// TIA Portal V20 program export: 1 tag tables, 5 data types, 30 data blocks, 9 code blocks (in call order from the OBs), 26 instance data blocks

VAR_GLOBAL   // PLC tag table "CentralFunctions"
END_VAR

TYPE "typeEmMotorStarterInterface"
// stored: Access Published
   STRUCT
      EMmotorstarter : Array[0.."NO_OF_EM"] of "typeMotorStarterInterface";
   END_STRUCT;
END_TYPE

TYPE "typeEt200SpMotorstarterInterfaceHmi"
// stored: Access Published
   STRUCT
      et200SpMotorstarterReadValue : Bool;   // read Value of MotorStarter
      et200SpNumberOfMotorstarters { ExternalWritable := 'False'} : USInt;   // Number of Motor Starters
      et200SpUnitMotorstarter : USInt := 1;   // Unit selected
      et200SpEMMotorstarter : USInt := 0;   // Equipment Module selected
      et200SpMotorstarterCurrent : Array[0.."NO_OF_ET200SPMOTORSTARTER"] of Real;   // Aktuelle Werte / Current values
      et200SpMotorstarterInputs : Array[0.."NO_OF_ET200SPMOTORSTARTER"] of "LSicar_typeMotorstarterIn";   // Motorstarter Data Inputs HMI
      et200SpMotorstarterOutputs : Array[0.."NO_OF_ET200SPMOTORSTARTER"] of "LSicar_typeMotorstarterOut";   // Motorstarter Data Outputs HMI
   END_STRUCT;
END_TYPE

TYPE "typeMotorStarterInterface"
// stored: Access Published
   STRUCT
      et200SpMotorstarterCurrent : Array[0.."NO_OF_ET200SPMOTORSTARTER"] of Real;   // Aktuelle Werte / Current values
      et200SpMotorstarterInputs : Array[0.."NO_OF_ET200SPMOTORSTARTER"] of "LSicar_typeMotorstarterIn";   // Motorstarter Data Inputs HMI
      et200SpMotorstarterOutputs : Array[0.."NO_OF_ET200SPMOTORSTARTER"] of "LSicar_typeMotorstarterOut";   // Motorstarter Data Outputs HMI
   END_STRUCT;
END_TYPE

TYPE "typeIdentMvHmi"
// stored: Access Published
   STRUCT
      selectedUnit : USInt;
      selectedEM : USInt;
      mvReaderId : USInt;   // MV Reader ID
      numberOfMv : USInt;   // Anzahl der MV Antriebe / Number of used MV readers
      mvReader : Array[0.."NO_OF_MV_IDENT_DEVICES"] of "LSicar_typeIdentInterfaceHmi";   // MV Reader
   END_STRUCT;
END_TYPE

TYPE "typeEMIdentRf"
// stored: Access Published
   STRUCT
      identRfEM : Array[0.."NO_OF_EM"] of "typeIdentRfHmi";
   END_STRUCT;
END_TYPE

DATA_BLOCK "TestTempDB"   // DB502
// stored: MemoryReserve 100
   VAR
      TempBool : Array[0..100] of Bool;
   END_VAR
BEGIN
END_DATA_BLOCK

DATA_BLOCK "Simulation"   // DB203
TITLE = Simulation
// Simulation data
// stored: MemoryReserve 100
   VAR
      simHmiRotaryAxis : Array[0..49] of "LER_typeSimRotaryAxis";
      simHmiLinearAxis : Array[0..49] of "LER_typeSimLinearAxis";
      data : "LAF_typeSimulation";
   END_VAR
BEGIN
   data.simitActive := FALSE;
   data.simulationActiveHmi := TRUE;
   data.showSimulationButtonHmi := TRUE;
END_DATA_BLOCK

DATA_BLOCK "ProdDataInterfaceHmi"   // DB53
TITLE = HMI und Anwender Schnittstelle für Produktionsdaten / HMI and user interface for production data
AUTHOR : SICAR
FAMILY : ProdData
// FUNKTIONSBESCHREIBUNG: 
// Der Baustein beinhaltet alle Informationen zum und vom HMI, sowie die Anwenderschnittstellen für die Produktionsdaten
// Weitere Hinweise: siehe SICAR anwenderdefinierte Dokumentation / SICAR Online-Hilfe.
// DESCRIPTION OF FUNCTIONS:
// stored: MemoryReserve 100
   VAR RETAIN
      numberOfDataSets : "LSicar_typeNumberOfDataSets";   // Anzahl konfigurierter Datensätze / Number of configured data sets
   END_VAR
   VAR
      colorCodeLimitSummary : UInt := 0;   // Gesamt Status Grenzwerte / Overall status Limit values
      colorCodeLimitSelButton : Array[0..8] of UInt;   // Farbcode für Datensatz Anwahl Button (Grenzwerte) / Color code for data set select button (Limit values)
   END_VAR
   VAR RETAIN
      limitValueDataSetSel : Int := 1;   // Angwaehlter Datensatz Grenzwerte / selected data set limit values
      limitDataSet : Array[0.."NO_DATASETS_LIMITVALUES"] of "LSicar_typeLimitValue";   // Datensätze Grenzwerte / Data sets limit .values
      cycleTimerDataSetSel : Int := 1;   // Angewaehlter Datensatz Taktzeiten / selected data set cycle timer
      cycleTimerDataSet : Array[0.."NO_DATASETS_CYCLETIMER"] of "LSicar_typeCycleTimer";   // Datensätze Taktzeiten / Data sets cycle timer
      counterDataSetSel : Int := 1;   // Angewählter Datensatz Zaehler / selected data set counter
      counterDataSet : Array[0.."NO_DATASETS_COUNTER"] of "LSicar_typeCounter";   // Datensätze Zähler / Data sets counter
      shiftCounterDataSetSel : Int := 1;   // Angewaehlter Datensatz Schichtzaehler / selected data set shift counter
      shiftCounterDataSet : Array[0.."NO_DATASETS_SHIFTCOUNTER"] of "LSicar_typeShiftCounter";   // Datensätze Schichtzähler / Data sets shift counter
      shiftCountOeeDataSetSel : Int := 1;   // Angewaehlter Datensatz OEE / selected data set OEE
      shiftCounterOeeDataSet : Array[0.."NO_DATASETS_SHIFTCOUNTER"] of "LSicar_typeShiftCounterOee";   // Datensätze Schichtzähler OEE / Data sets shift counter OEE
   END_VAR
BEGIN
   numberOfDataSets.limitValues := 2;
   numberOfDataSets.cycleTimer := 2;
   numberOfDataSets."counter" := 2;
   numberOfDataSets.shiftCounter := 2;
   colorCodeLimitSelButton[0..8] := 0;
   limitDataSet[0].targetValue[0..10] := 0;
   limitDataSet[1].targetValue[0..10] := 0;
   limitDataSet[2].targetValue[0..10] := 0;
   limitDataSet[0].prewarnValue[0..10] := 0;
   limitDataSet[1].prewarnValue[0..10] := 0;
   limitDataSet[2].prewarnValue[0..10] := 0;
   limitDataSet[0].remainValue[0..10] := 0;
   limitDataSet[1].remainValue[0..10] := 0;
   limitDataSet[2].remainValue[0..10] := 0;
   limitDataSet[0].control[0..10].count := FALSE;
   limitDataSet[1].control[0..10].count := FALSE;
   limitDataSet[2].control[0..10].count := FALSE;
   limitDataSet[0].control[0..10].set := FALSE;
   limitDataSet[1].control[0..10].set := FALSE;
   limitDataSet[2].control[0..10].set := FALSE;
   limitDataSet[0].control[0..10].prewarn := FALSE;
   limitDataSet[1].control[0..10].prewarn := FALSE;
   limitDataSet[2].control[0..10].prewarn := FALSE;
   limitDataSet[0].control[0..10].alarm := FALSE;
   limitDataSet[1].control[0..10].alarm := FALSE;
   limitDataSet[2].control[0..10].alarm := FALSE;
   limitDataSet[0].textListValue[0..10] := 0;
   limitDataSet[1].textListValue[0..10] := 0;
   limitDataSet[2].textListValue[0..10] := 0;
   limitDataSet[0..2].userInterfaceVisibility := 16#0000_0000;
   limitDataSet[0].colorCodeAlarmPrewarn[0..10] := 0;
   limitDataSet[1].colorCodeAlarmPrewarn[0..10] := 0;
   limitDataSet[2].colorCodeAlarmPrewarn[0..10] := 0;
   limitDataSet[0..2].indexSelectedLimitValue := 0;
   limitDataSet[0..2].divButton := 16#00;
   limitDataSet[0..2].visibility := 16#0000_0000;
   cycleTimerDataSet[0].targetValue[0..20] := 0;
   cycleTimerDataSet[1].targetValue[0..20] := 0;
   cycleTimerDataSet[2].targetValue[0..20] := 0;
   cycleTimerDataSet[0].currentValue[0..20] := 0;
   cycleTimerDataSet[1].currentValue[0..20] := 0;
   cycleTimerDataSet[2].currentValue[0..20] := 0;
   cycleTimerDataSet[0].averageValue[0..20] := 0;
   cycleTimerDataSet[1].averageValue[0..20] := 0;
   cycleTimerDataSet[2].averageValue[0..20] := 0;
   cycleTimerDataSet[0].counts[0..20] := 0;
   cycleTimerDataSet[1].counts[0..20] := 0;
   cycleTimerDataSet[2].counts[0..20] := 0;
   cycleTimerDataSet[0].measureActive[0..20] := 0;
   cycleTimerDataSet[1].measureActive[0..20] := 0;
   cycleTimerDataSet[2].measureActive[0..20] := 0;
   cycleTimerDataSet[0].control[0..20].run := FALSE;
   cycleTimerDataSet[1].control[0..20].run := FALSE;
   cycleTimerDataSet[2].control[0..20].run := FALSE;
   cycleTimerDataSet[0].control[0..20].hold := FALSE;
   cycleTimerDataSet[1].control[0..20].hold := FALSE;
   cycleTimerDataSet[2].control[0..20].hold := FALSE;
   cycleTimerDataSet[0].control[0..20].reset := FALSE;
   cycleTimerDataSet[1].control[0..20].reset := FALSE;
   cycleTimerDataSet[2].control[0..20].reset := FALSE;
   cycleTimerDataSet[0].textListValue[0..20] := 0;
   cycleTimerDataSet[1].textListValue[0..20] := 0;
   cycleTimerDataSet[2].textListValue[0..20] := 0;
   cycleTimerDataSet[0..2].userInterfaceVisibility := 16#0000_0000;
   cycleTimerDataSet[0..2].resetAverageAllExt := FALSE;
   cycleTimerDataSet[0..2].indexSelectedTimer := 0;
   cycleTimerDataSet[0..2].divButton := 16#00;
   cycleTimerDataSet[0..2].visibility := 16#0000_0000;
   counterDataSet[0].currentValue[0..20] := 0;
   counterDataSet[1].currentValue[0..20] := 0;
   counterDataSet[2].currentValue[0..20] := 0;
   counterDataSet[0].control[0..20].countUp := FALSE;
   counterDataSet[1].control[0..20].countUp := FALSE;
   counterDataSet[2].control[0..20].countUp := FALSE;
   counterDataSet[0].control[0..20].countDown := FALSE;
   counterDataSet[1].control[0..20].countDown := FALSE;
   counterDataSet[2].control[0..20].countDown := FALSE;
   counterDataSet[0].control[0..20].reset := FALSE;
   counterDataSet[1].control[0..20].reset := FALSE;
   counterDataSet[2].control[0..20].reset := FALSE;
   counterDataSet[0].textListValue[0..20] := 0;
   counterDataSet[1].textListValue[0..20] := 0;
   counterDataSet[2].textListValue[0..20] := 0;
   counterDataSet[0].userInterfaceVisibility := 16#0000_0000;
   counterDataSet[1].userInterfaceVisibility := 16#0000_0007;
   counterDataSet[2].userInterfaceVisibility := 16#0000_0003;
   counterDataSet[0..2].resetAllExt := FALSE;
   counterDataSet[0..2].indexSelectedCounter := 0;
   counterDataSet[0..2].divButton := 16#00;
   counterDataSet[0..2].visibility := 16#0000_0000;
   shiftCounterDataSet[0].currentShiftValue.partsTarget[0..10] := 0;
   shiftCounterDataSet[1].currentShiftValue.partsTarget[0..10] := 0;
   shiftCounterDataSet[2].currentShiftValue.partsTarget[0..10] := 0;
   shiftCounterDataSet[0].currentShiftValue.partsCurrent[0..10] := 0;
   shiftCounterDataSet[1].currentShiftValue.partsCurrent[0..10] := 0;
   shiftCounterDataSet[2].currentShiftValue.partsCurrent[0..10] := 0;
   shiftCounterDataSet[0].previousShiftValue.partsTarget[0..10] := 0;
   shiftCounterDataSet[1].previousShiftValue.partsTarget[0..10] := 0;
   shiftCounterDataSet[2].previousShiftValue.partsTarget[0..10] := 0;
   shiftCounterDataSet[0].previousShiftValue.partsCurrent[0..10] := 0;
   shiftCounterDataSet[1].previousShiftValue.partsCurrent[0..10] := 0;
   shiftCounterDataSet[2].previousShiftValue.partsCurrent[0..10] := 0;
   shiftCounterDataSet[0].penultimateShiftValue.partsTarget[0..10] := 0;
   shiftCounterDataSet[1].penultimateShiftValue.partsTarget[0..10] := 0;
   shiftCounterDataSet[2].penultimateShiftValue.partsTarget[0..10] := 0;
   shiftCounterDataSet[0].penultimateShiftValue.partsCurrent[0..10] := 0;
   shiftCounterDataSet[1].penultimateShiftValue.partsCurrent[0..10] := 0;
   shiftCounterDataSet[2].penultimateShiftValue.partsCurrent[0..10] := 0;
   shiftCounterDataSet[0].countPartsCurrent[0..10] := FALSE;
   shiftCounterDataSet[1].countPartsCurrent[0..10] := FALSE;
   shiftCounterDataSet[2].countPartsCurrent[0..10] := FALSE;
   shiftCounterDataSet[0].textListValue[0..10] := 0;
   shiftCounterDataSet[1].textListValue[0..10] := 0;
   shiftCounterDataSet[2].textListValue[0..10] := 0;
   shiftCounterDataSet[0..2].userInterfaceVisibility := 16#0000_0000;
   shiftCounterDataSet[0..2].resetAllExt := FALSE;
   shiftCounterDataSet[0..2].divButton := 16#00;
   shiftCounterDataSet[0..2].visibility := 16#0000_0000;
   shiftCounterOeeDataSet[0].currentShiftValue.oee[0..10] := 0.0;
   shiftCounterOeeDataSet[1].currentShiftValue.oee[0..10] := 0.0;
   shiftCounterOeeDataSet[2].currentShiftValue.oee[0..10] := 0.0;
   shiftCounterOeeDataSet[0].currentShiftValue.trend[0..10] := 0;
   shiftCounterOeeDataSet[1].currentShiftValue.trend[0..10] := 0;
   shiftCounterOeeDataSet[2].currentShiftValue.trend[0..10] := 0;
   shiftCounterOeeDataSet[0].currentShiftValue.partsTarget[0..10] := 0;
   shiftCounterOeeDataSet[1].currentShiftValue.partsTarget[0..10] := 0;
   shiftCounterOeeDataSet[2].currentShiftValue.partsTarget[0..10] := 0;
   shiftCounterOeeDataSet[0].currentShiftValue.partsCurrent[0..10] := 0;
   shiftCounterOeeDataSet[1].currentShiftValue.partsCurrent[0..10] := 0;
   shiftCounterOeeDataSet[2].currentShiftValue.partsCurrent[0..10] := 0;
   shiftCounterOeeDataSet[0].currentShiftValue.partsCurrentOk[0..10] := 0;
   shiftCounterOeeDataSet[1].currentShiftValue.partsCurrentOk[0..10] := 0;
   shiftCounterOeeDataSet[2].currentShiftValue.partsCurrentOk[0..10] := 0;
   shiftCounterOeeDataSet[0].previousShiftValue.oee[0..10] := 0.0;
   shiftCounterOeeDataSet[1].previousShiftValue.oee[0..10] := 0.0;
   shiftCounterOeeDataSet[2].previousShiftValue.oee[0..10] := 0.0;
   shiftCounterOeeDataSet[0].previousShiftValue.trend[0..10] := 0;
   shiftCounterOeeDataSet[1].previousShiftValue.trend[0..10] := 0;
   shiftCounterOeeDataSet[2].previousShiftValue.trend[0..10] := 0;
   shiftCounterOeeDataSet[0].previousShiftValue.partsTarget[0..10] := 0;
   shiftCounterOeeDataSet[1].previousShiftValue.partsTarget[0..10] := 0;
   shiftCounterOeeDataSet[2].previousShiftValue.partsTarget[0..10] := 0;
   shiftCounterOeeDataSet[0].previousShiftValue.partsCurrent[0..10] := 0;
   shiftCounterOeeDataSet[1].previousShiftValue.partsCurrent[0..10] := 0;
   shiftCounterOeeDataSet[2].previousShiftValue.partsCurrent[0..10] := 0;
   shiftCounterOeeDataSet[0].previousShiftValue.partsCurrentOk[0..10] := 0;
   shiftCounterOeeDataSet[1].previousShiftValue.partsCurrentOk[0..10] := 0;
   shiftCounterOeeDataSet[2].previousShiftValue.partsCurrentOk[0..10] := 0;
   shiftCounterOeeDataSet[0].penultimateShiftValue.oee[0..10] := 0.0;
   shiftCounterOeeDataSet[1].penultimateShiftValue.oee[0..10] := 0.0;
   shiftCounterOeeDataSet[2].penultimateShiftValue.oee[0..10] := 0.0;
   shiftCounterOeeDataSet[0].penultimateShiftValue.trend[0..10] := 0;
   shiftCounterOeeDataSet[1].penultimateShiftValue.trend[0..10] := 0;
   shiftCounterOeeDataSet[2].penultimateShiftValue.trend[0..10] := 0;
   shiftCounterOeeDataSet[0].penultimateShiftValue.partsTarget[0..10] := 0;
   shiftCounterOeeDataSet[1].penultimateShiftValue.partsTarget[0..10] := 0;
   shiftCounterOeeDataSet[2].penultimateShiftValue.partsTarget[0..10] := 0;
   shiftCounterOeeDataSet[0].penultimateShiftValue.partsCurrent[0..10] := 0;
   shiftCounterOeeDataSet[1].penultimateShiftValue.partsCurrent[0..10] := 0;
   shiftCounterOeeDataSet[2].penultimateShiftValue.partsCurrent[0..10] := 0;
   shiftCounterOeeDataSet[0].penultimateShiftValue.partsCurrentOk[0..10] := 0;
   shiftCounterOeeDataSet[1].penultimateShiftValue.partsCurrentOk[0..10] := 0;
   shiftCounterOeeDataSet[2].penultimateShiftValue.partsCurrentOk[0..10] := 0;
   shiftCounterOeeDataSet[0].countPartsCurrent[0..10] := FALSE;
   shiftCounterOeeDataSet[1].countPartsCurrent[0..10] := FALSE;
   shiftCounterOeeDataSet[2].countPartsCurrent[0..10] := FALSE;
   shiftCounterOeeDataSet[0].countPartsCurrentOk[0..10] := FALSE;
   shiftCounterOeeDataSet[1].countPartsCurrentOk[0..10] := FALSE;
   shiftCounterOeeDataSet[2].countPartsCurrentOk[0..10] := FALSE;
   shiftCounterOeeDataSet[0].textListValue[0..10] := 0;
   shiftCounterOeeDataSet[1].textListValue[0..10] := 0;
   shiftCounterOeeDataSet[2].textListValue[0..10] := 0;
   shiftCounterOeeDataSet[0..2].userInterfaceVisibility := 16#0000_0000;
   shiftCounterOeeDataSet[0..2].resetAllExt := FALSE;
   shiftCounterOeeDataSet[0..2].divButton := 16#00;
   shiftCounterOeeDataSet[0..2].visibility := 16#0000_0000;
END_DATA_BLOCK

DATA_BLOCK "ShiftTimesList"   // DB52
TITLE = Shifttimes / Shift times
{ DB_Accessible_From_OPC_UA := 'FALSE' }
AUTHOR : SICAR
FAMILY : Shiftmodel
// Schichtzeiten Liste / Shift times List
// stored: DBAccessibleFromOPCUA false, MemoryReserve 100
   VAR
      list { ExternalAccessible := 'False'; ExternalVisible := 'False'; ExternalWritable := 'False'} : Array[0..10] of "LSicar_typeShiftmodTime1DaySel";   // Schichtmodel Liste / Shiftmodel list
   END_VAR
BEGIN
   list[0..2].listValidFor.sunday := FALSE;
   list[3].listValidFor.sunday := TRUE;
   list[4..10].listValidFor.sunday := FALSE;
   list[0].listValidFor.monday := FALSE;
   list[1..3].listValidFor.monday := TRUE;
   list[4..10].listValidFor.monday := FALSE;
   list[0].listValidFor.tuesday := FALSE;
   list[1..3].listValidFor.tuesday := TRUE;
   list[4..10].listValidFor.tuesday := FALSE;
   list[0].listValidFor.wednesday := FALSE;
   list[1..3].listValidFor.wednesday := TRUE;
   list[4..10].listValidFor.wednesday := FALSE;
   list[0].listValidFor.thursday := FALSE;
   list[1..3].listValidFor.thursday := TRUE;
   list[4..10].listValidFor.thursday := FALSE;
   list[0].listValidFor.friday := FALSE;
   list[1].listValidFor.friday := TRUE;
   list[2].listValidFor.friday := FALSE;
   list[3].listValidFor.friday := TRUE;
   list[4..10].listValidFor.friday := FALSE;
   list[0..2].listValidFor.saturday := FALSE;
   list[3].listValidFor.saturday := TRUE;
   list[4..10].listValidFor.saturday := FALSE;
   list[0].shift[0..3].endCircuitTime := TOD#00:00:00;
   list[1].shift[0].endCircuitTime := TOD#00:00:00;
   list[1].shift[1].endCircuitTime := TOD#05:57:00;
   list[1].shift[2].endCircuitTime := TOD#13:57:00;
   list[1].shift[3].endCircuitTime := TOD#21:57:00;
   list[2].shift[0].endCircuitTime := TOD#00:00:00;
   list[2].shift[1].endCircuitTime := TOD#04:57:00;
   list[2].shift[2].endCircuitTime := TOD#14:27:00;
   list[2].shift[3].endCircuitTime := TOD#00:00:00;
   list[3].shift[0].endCircuitTime := TOD#00:00:00;
   list[3].shift[1].endCircuitTime := TOD#05:57:00;
   list[3].shift[2].endCircuitTime := TOD#14:27:00;
   list[3].shift[3].endCircuitTime := TOD#22:57:00;
   list[4].shift[0..3].endCircuitTime := TOD#00:00:00;
   list[5].shift[0..3].endCircuitTime := TOD#00:00:00;
   list[6].shift[0..3].endCircuitTime := TOD#00:00:00;
   list[7].shift[0..3].endCircuitTime := TOD#00:00:00;
   list[8].shift[0..3].endCircuitTime := TOD#00:00:00;
   list[9].shift[0..3].endCircuitTime := TOD#00:00:00;
   list[10].shift[0..3].endCircuitTime := TOD#00:00:00;
   list[0].shift[0..3].start := TOD#00:00:00;
   list[1].shift[0].start := TOD#00:00:00;
   list[1].shift[1].start := TOD#06:00:00;
   list[1].shift[2].start := TOD#14:00:00;
   list[1].shift[3].start := TOD#22:00:00;
   list[2].shift[0].start := TOD#00:00:00;
   list[2].shift[1].start := TOD#05:00:00;
   list[2].shift[2].start := TOD#14:30:00;
   list[2].shift[3].start := TOD#00:00:00;
   list[3].shift[0].start := TOD#00:00:00;
   list[3].shift[1].start := TOD#06:00:00;
   list[3].shift[2].start := TOD#14:30:00;
   list[3].shift[3].start := TOD#23:00:00;
   list[4].shift[0..3].start := TOD#00:00:00;
   list[5].shift[0..3].start := TOD#00:00:00;
   list[6].shift[0..3].start := TOD#00:00:00;
   list[7].shift[0..3].start := TOD#00:00:00;
   list[8].shift[0..3].start := TOD#00:00:00;
   list[9].shift[0..3].start := TOD#00:00:00;
   list[10].shift[0..3].start := TOD#00:00:00;
   list[0].shift[0].break[0..4].start := TOD#00:00:00;
   list[0].shift[1].break[0..4].start := TOD#00:00:00;
   list[0].shift[2].break[0..4].start := TOD#00:00:00;
   list[0].shift[3].break[0..4].start := TOD#00:00:00;
   list[1].shift[0].break[0..4].start := TOD#00:00:00;
   list[1].shift[1].break[0].start := TOD#00:00:00;
   list[1].shift[1].break[1].start := TOD#08:00:00;
   list[1].shift[1].break[2].start := TOD#10:00:00;
   list[1].shift[1].break[3].start := TOD#12:00:00;
   list[1].shift[1].break[4].start := TOD#00:00:00;
   list[1].shift[2].break[0].start := TOD#00:00:00;
   list[1].shift[2].break[1].start := TOD#16:00:00;
   list[1].shift[2].break[2].start := TOD#18:00:00;
   list[1].shift[2].break[3].start := TOD#20:00:00;
   list[1].shift[2].break[4].start := TOD#00:00:00;
   list[1].shift[3].break[0..1].start := TOD#00:00:00;
   list[1].shift[3].break[2].start := TOD#02:00:00;
   list[1].shift[3].break[3].start := TOD#04:00:00;
   list[1].shift[3].break[4].start := TOD#00:00:00;
   list[2].shift[0].break[0..4].start := TOD#00:00:00;
   list[2].shift[1].break[0].start := TOD#00:00:00;
   list[2].shift[1].break[1].start := TOD#07:00:00;
   list[2].shift[1].break[2].start := TOD#09:00:00;
   list[2].shift[1].break[3].start := TOD#11:00:00;
   list[2].shift[1].break[4].start := TOD#13:00:00;
   list[2].shift[2].break[0].start := TOD#00:00:00;
   list[2].shift[2].break[1].start := TOD#16:30:00;
   list[2].shift[2].break[2].start := TOD#18:30:00;
   list[2].shift[2].break[3].start := TOD#20:30:00;
   list[2].shift[2].break[4].start := TOD#22:00:00;
   list[2].shift[3].break[0..4].start := TOD#00:00:00;
   list[3].shift[0].break[0..4].start := TOD#00:00:00;
   list[3].shift[1].break[0].start := TOD#00:00:00;
   list[3].shift[1].break[1].start := TOD#08:00:00;
   list[3].shift[1].break[2].start := TOD#10:00:00;
   list[3].shift[1].break[3].start := TOD#11:30:00;
   list[3].shift[1].break[4].start := TOD#12:30:00;
   list[3].shift[2].break[0].start := TOD#00:00:00;
   list[3].shift[2].break[1].start := TOD#16:00:00;
   list[3].shift[2].break[2].start := TOD#18:00:00;
   list[3].shift[2].break[3].start := TOD#19:30:00;
   list[3].shift[2].break[4].start := TOD#20:30:00;
   list[3].shift[3].break[0..1].start := TOD#00:00:00;
   list[3].shift[3].break[2].start := TOD#02:00:00;
   list[3].shift[3].break[3].start := TOD#03:30:00;
   list[3].shift[3].break[4].start := TOD#04:30:00;
   list[4].shift[0].break[0..4].start := TOD#00:00:00;
   list[4].shift[1].break[0..4].start := TOD#00:00:00;
   list[4].shift[2].break[0..4].start := TOD#00:00:00;
   list[4].shift[3].break[0..4].start := TOD#00:00:00;
   list[5].shift[0].break[0..4].start := TOD#00:00:00;
   list[5].shift[1].break[0..4].start := TOD#00:00:00;
   list[5].shift[2].break[0..4].start := TOD#00:00:00;
   list[5].shift[3].break[0..4].start := TOD#00:00:00;
   list[6].shift[0].break[0..4].start := TOD#00:00:00;
   list[6].shift[1].break[0..4].start := TOD#00:00:00;
   list[6].shift[2].break[0..4].start := TOD#00:00:00;
   list[6].shift[3].break[0..4].start := TOD#00:00:00;
   list[7].shift[0].break[0..4].start := TOD#00:00:00;
   list[7].shift[1].break[0..4].start := TOD#00:00:00;
   list[7].shift[2].break[0..4].start := TOD#00:00:00;
   list[7].shift[3].break[0..4].start := TOD#00:00:00;
   list[8].shift[0].break[0..4].start := TOD#00:00:00;
   list[8].shift[1].break[0..4].start := TOD#00:00:00;
   list[8].shift[2].break[0..4].start := TOD#00:00:00;
   list[8].shift[3].break[0..4].start := TOD#00:00:00;
   list[9].shift[0].break[0..4].start := TOD#00:00:00;
   list[9].shift[1].break[0..4].start := TOD#00:00:00;
   list[9].shift[2].break[0..4].start := TOD#00:00:00;
   list[9].shift[3].break[0..4].start := TOD#00:00:00;
   list[10].shift[0].break[0..4].start := TOD#00:00:00;
   list[10].shift[1].break[0..4].start := TOD#00:00:00;
   list[10].shift[2].break[0..4].start := TOD#00:00:00;
   list[10].shift[3].break[0..4].start := TOD#00:00:00;
   list[0].shift[0].break[0..4].startCircuitTime := TOD#00:00:00;
   list[0].shift[1].break[0..4].startCircuitTime := TOD#00:00:00;
   list[0].shift[2].break[0..4].startCircuitTime := TOD#00:00:00;
   list[0].shift[3].break[0..4].startCircuitTime := TOD#00:00:00;
   list[1].shift[0].break[0..4].startCircuitTime := TOD#00:00:00;
   list[1].shift[1].break[0].startCircuitTime := TOD#00:00:00;
   list[1].shift[1].break[1].startCircuitTime := TOD#08:02:00;
   list[1].shift[1].break[2].startCircuitTime := TOD#00:00:00;
   list[1].shift[1].break[3].startCircuitTime := TOD#12:02:00;
   list[1].shift[1].break[4].startCircuitTime := TOD#00:00:00;
   list[1].shift[2].break[0].startCircuitTime := TOD#00:00:00;
   list[1].shift[2].break[1].startCircuitTime := TOD#16:02:00;
   list[1].shift[2].break[2].startCircuitTime := TOD#00:00:00;
   list[1].shift[2].break[3].startCircuitTime := TOD#20:02:00;
   list[1].shift[2].break[4].startCircuitTime := TOD#00:00:00;
   list[1].shift[3].break[0].startCircuitTime := TOD#00:00:00;
   list[1].shift[3].break[1].startCircuitTime := TOD#00:02:00;
   list[1].shift[3].break[2].startCircuitTime := TOD#00:00:00;
   list[1].shift[3].break[3].startCircuitTime := TOD#04:02:00;
   list[1].shift[3].break[4].startCircuitTime := TOD#00:00:00;
   list[2].shift[0].break[0..4].startCircuitTime := TOD#00:00:00;
   list[2].shift[1].break[0].startCircuitTime := TOD#00:00:00;
   list[2].shift[1].break[1].startCircuitTime := TOD#07:02:00;
   list[2].shift[1].break[2].startCircuitTime := TOD#00:00:00;
   list[2].shift[1].break[3].startCircuitTime := TOD#11:02:00;
   list[2].shift[1].break[4].startCircuitTime := TOD#13:02:00;
   list[2].shift[2].break[0].startCircuitTime := TOD#00:00:00;
   list[2].shift[2].break[1].startCircuitTime := TOD#16:32:00;
   list[2].shift[2].break[2].startCircuitTime := TOD#00:00:00;
   list[2].shift[2].break[3].startCircuitTime := TOD#20:32:00;
   list[2].shift[2].break[4].startCircuitTime := TOD#22:02:00;
   list[2].shift[3].break[0..4].startCircuitTime := TOD#00:00:00;
   list[3].shift[0].break[0..4].startCircuitTime := TOD#00:00:00;
   list[3].shift[1].break[0..1].startCircuitTime := TOD#00:00:00;
   list[3].shift[1].break[2].startCircuitTime := TOD#10:02:00;
   list[3].shift[1].break[3].startCircuitTime := TOD#00:00:00;
   list[3].shift[1].break[4].startCircuitTime := TOD#12:32:00;
   list[3].shift[2].break[0..1].startCircuitTime := TOD#00:00:00;
   list[3].shift[2].break[2].startCircuitTime := TOD#18:02:00;
   list[3].shift[2].break[3].startCircuitTime := TOD#00:00:00;
   list[3].shift[2].break[4].startCircuitTime := TOD#20:32:00;
   list[3].shift[3].break[0..1].startCircuitTime := TOD#00:00:00;
   list[3].shift[3].break[2].startCircuitTime := TOD#02:02:00;
   list[3].shift[3].break[3..4].startCircuitTime := TOD#00:00:00;
   list[4].shift[0].break[0..4].startCircuitTime := TOD#00:00:00;
   list[4].shift[1].break[0..4].startCircuitTime := TOD#00:00:00;
   list[4].shift[2].break[0..4].startCircuitTime := TOD#00:00:00;
   list[4].shift[3].break[0..4].startCircuitTime := TOD#00:00:00;
   list[5].shift[0].break[0..4].startCircuitTime := TOD#00:00:00;
   list[5].shift[1].break[0..4].startCircuitTime := TOD#00:00:00;
   list[5].shift[2].break[0..4].startCircuitTime := TOD#00:00:00;
   list[5].shift[3].break[0..4].startCircuitTime := TOD#00:00:00;
   list[6].shift[0].break[0..4].startCircuitTime := TOD#00:00:00;
   list[6].shift[1].break[0..4].startCircuitTime := TOD#00:00:00;
   list[6].shift[2].break[0..4].startCircuitTime := TOD#00:00:00;
   list[6].shift[3].break[0..4].startCircuitTime := TOD#00:00:00;
   list[7].shift[0].break[0..4].startCircuitTime := TOD#00:00:00;
   list[7].shift[1].break[0..4].startCircuitTime := TOD#00:00:00;
   list[7].shift[2].break[0..4].startCircuitTime := TOD#00:00:00;
   list[7].shift[3].break[0..4].startCircuitTime := TOD#00:00:00;
   list[8].shift[0].break[0..4].startCircuitTime := TOD#00:00:00;
   list[8].shift[1].break[0..4].startCircuitTime := TOD#00:00:00;
   list[8].shift[2].break[0..4].startCircuitTime := TOD#00:00:00;
   list[8].shift[3].break[0..4].startCircuitTime := TOD#00:00:00;
   list[9].shift[0].break[0..4].startCircuitTime := TOD#00:00:00;
   list[9].shift[1].break[0..4].startCircuitTime := TOD#00:00:00;
   list[9].shift[2].break[0..4].startCircuitTime := TOD#00:00:00;
   list[9].shift[3].break[0..4].startCircuitTime := TOD#00:00:00;
   list[10].shift[0].break[0..4].startCircuitTime := TOD#00:00:00;
   list[10].shift[1].break[0..4].startCircuitTime := TOD#00:00:00;
   list[10].shift[2].break[0..4].startCircuitTime := TOD#00:00:00;
   list[10].shift[3].break[0..4].startCircuitTime := TOD#00:00:00;
   list[0].shift[0].break[0..4].endCircuitTime := TOD#00:00:00;
   list[0].shift[1].break[0..4].endCircuitTime := TOD#00:00:00;
   list[0].shift[2].break[0..4].endCircuitTime := TOD#00:00:00;
   list[0].shift[3].break[0..4].endCircuitTime := TOD#00:00:00;
   list[1].shift[0].break[0..4].endCircuitTime := TOD#00:00:00;
   list[1].shift[1].break[0].endCircuitTime := TOD#00:00:00;
   list[1].shift[1].break[1].endCircuitTime := TOD#08:13:00;
   list[1].shift[1].break[2].endCircuitTime := TOD#00:00:00;
   list[1].shift[1].break[3].endCircuitTime := TOD#12:13:00;
   list[1].shift[1].break[4].endCircuitTime := TOD#00:00:00;
   list[1].shift[2].break[0].endCircuitTime := TOD#00:00:00;
   list[1].shift[2].break[1].endCircuitTime := TOD#16:13:00;
   list[1].shift[2].break[2].endCircuitTime := TOD#00:00:00;
   list[1].shift[2].break[3].endCircuitTime := TOD#20:13:00;
   list[1].shift[2].break[4].endCircuitTime := TOD#00:00:00;
   list[1].shift[3].break[0].endCircuitTime := TOD#00:00:00;
   list[1].shift[3].break[1].endCircuitTime := TOD#00:13:00;
   list[1].shift[3].break[2].endCircuitTime := TOD#00:00:00;
   list[1].shift[3].break[3].endCircuitTime := TOD#04:13:00;
   list[1].shift[3].break[4].endCircuitTime := TOD#00:00:00;
   list[2].shift[0].break[0..4].endCircuitTime := TOD#00:00:00;
   list[2].shift[1].break[0].endCircuitTime := TOD#00:00:00;
   list[2].shift[1].break[1].endCircuitTime := TOD#07:13:00;
   list[2].shift[1].break[2].endCircuitTime := TOD#00:00:00;
   list[2].shift[1].break[3].endCircuitTime := TOD#11:13:00;
   list[2].shift[1].break[4].endCircuitTime := TOD#13:13:00;
   list[2].shift[2].break[0].endCircuitTime := TOD#00:00:00;
   list[2].shift[2].break[1].endCircuitTime := TOD#16:43:00;
   list[2].shift[2].break[2].endCircuitTime := TOD#00:00:00;
   list[2].shift[2].break[3].endCircuitTime := TOD#20:43:00;
   list[2].shift[2].break[4].endCircuitTime := TOD#22:13:00;
   list[2].shift[3].break[0..4].endCircuitTime := TOD#00:00:00;
   list[3].shift[0].break[0..4].endCircuitTime := TOD#00:00:00;
   list[3].shift[1].break[0..1].endCircuitTime := TOD#00:00:00;
   list[3].shift[1].break[2].endCircuitTime := TOD#10:13:00;
   list[3].shift[1].break[3].endCircuitTime := TOD#00:00:00;
   list[3].shift[1].break[4].endCircuitTime := TOD#12:43:00;
   list[3].shift[2].break[0..1].endCircuitTime := TOD#00:00:00;
   list[3].shift[2].break[2].endCircuitTime := TOD#18:13:00;
   list[3].shift[2].break[3].endCircuitTime := TOD#00:00:00;
   list[3].shift[2].break[4].endCircuitTime := TOD#20:43:00;
   list[3].shift[3].break[0..1].endCircuitTime := TOD#00:00:00;
   list[3].shift[3].break[2].endCircuitTime := TOD#02:13:00;
   list[3].shift[3].break[3..4].endCircuitTime := TOD#00:00:00;
   list[4].shift[0].break[0..4].endCircuitTime := TOD#00:00:00;
   list[4].shift[1].break[0..4].endCircuitTime := TOD#00:00:00;
   list[4].shift[2].break[0..4].endCircuitTime := TOD#00:00:00;
   list[4].shift[3].break[0..4].endCircuitTime := TOD#00:00:00;
   list[5].shift[0].break[0..4].endCircuitTime := TOD#00:00:00;
   list[5].shift[1].break[0..4].endCircuitTime := TOD#00:00:00;
   list[5].shift[2].break[0..4].endCircuitTime := TOD#00:00:00;
   list[5].shift[3].break[0..4].endCircuitTime := TOD#00:00:00;
   list[6].shift[0].break[0..4].endCircuitTime := TOD#00:00:00;
   list[6].shift[1].break[0..4].endCircuitTime := TOD#00:00:00;
   list[6].shift[2].break[0..4].endCircuitTime := TOD#00:00:00;
   list[6].shift[3].break[0..4].endCircuitTime := TOD#00:00:00;
   list[7].shift[0].break[0..4].endCircuitTime := TOD#00:00:00;
   list[7].shift[1].break[0..4].endCircuitTime := TOD#00:00:00;
   list[7].shift[2].break[0..4].endCircuitTime := TOD#00:00:00;
   list[7].shift[3].break[0..4].endCircuitTime := TOD#00:00:00;
   list[8].shift[0].break[0..4].endCircuitTime := TOD#00:00:00;
   list[8].shift[1].break[0..4].endCircuitTime := TOD#00:00:00;
   list[8].shift[2].break[0..4].endCircuitTime := TOD#00:00:00;
   list[8].shift[3].break[0..4].endCircuitTime := TOD#00:00:00;
   list[9].shift[0].break[0..4].endCircuitTime := TOD#00:00:00;
   list[9].shift[1].break[0..4].endCircuitTime := TOD#00:00:00;
   list[9].shift[2].break[0..4].endCircuitTime := TOD#00:00:00;
   list[9].shift[3].break[0..4].endCircuitTime := TOD#00:00:00;
   list[10].shift[0].break[0..4].endCircuitTime := TOD#00:00:00;
   list[10].shift[1].break[0..4].endCircuitTime := TOD#00:00:00;
   list[10].shift[2].break[0..4].endCircuitTime := TOD#00:00:00;
   list[10].shift[3].break[0..4].endCircuitTime := TOD#00:00:00;
   list[0].shift[0].break[0..4].end := TOD#00:00:00;
   list[0].shift[1].break[0..4].end := TOD#00:00:00;
   list[0].shift[2].break[0..4].end := TOD#00:00:00;
   list[0].shift[3].break[0..4].end := TOD#00:00:00;
   list[1].shift[0].break[0..4].end := TOD#00:00:00;
   list[1].shift[1].break[0].end := TOD#00:00:00;
   list[1].shift[1].break[1].end := TOD#08:15:00;
   list[1].shift[1].break[2].end := TOD#10:10:00;
   list[1].shift[1].break[3].end := TOD#12:15:00;
   list[1].shift[1].break[4].end := TOD#00:00:00;
   list[1].shift[2].break[0].end := TOD#00:00:00;
   list[1].shift[2].break[1].end := TOD#16:15:00;
   list[1].shift[2].break[2].end := TOD#18:10:00;
   list[1].shift[2].break[3].end := TOD#20:15:00;
   list[1].shift[2].break[4].end := TOD#00:00:00;
   list[1].shift[3].break[0].end := TOD#00:00:00;
   list[1].shift[3].break[1].end := TOD#00:15:00;
   list[1].shift[3].break[2].end := TOD#02:10:00;
   list[1].shift[3].break[3].end := TOD#04:15:00;
   list[1].shift[3].break[4].end := TOD#00:00:00;
   list[2].shift[0].break[0..4].end := TOD#00:00:00;
   list[2].shift[1].break[0].end := TOD#00:00:00;
   list[2].shift[1].break[1].end := TOD#07:15:00;
   list[2].shift[1].break[2].end := TOD#09:10:00;
   list[2].shift[1].break[3].end := TOD#11:15:00;
   list[2].shift[1].break[4].end := TOD#13:15:00;
   list[2].shift[2].break[0].end := TOD#00:00:00;
   list[2].shift[2].break[1].end := TOD#16:45:00;
   list[2].shift[2].break[2].end := TOD#18:40:00;
   list[2].shift[2].break[3].end := TOD#20:45:00;
   list[2].shift[2].break[4].end := TOD#22:15:00;
   list[2].shift[3].break[0..4].end := TOD#00:00:00;
   list[3].shift[0].break[0..4].end := TOD#00:00:00;
   list[3].shift[1].break[0].end := TOD#00:00:00;
   list[3].shift[1].break[1].end := TOD#08:10:00;
   list[3].shift[1].break[2].end := TOD#10:15:00;
   list[3].shift[1].break[3].end := TOD#11:40:00;
   list[3].shift[1].break[4].end := TOD#12:45:00;
   list[3].shift[2].break[0].end := TOD#00:00:00;
   list[3].shift[2].break[1].end := TOD#16:10:00;
   list[3].shift[2].break[2].end := TOD#18:15:00;
   list[3].shift[2].break[3].end := TOD#19:40:00;
   list[3].shift[2].break[4].end := TOD#20:45:00;
   list[3].shift[3].break[0].end := TOD#00:00:00;
   list[3].shift[3].break[1].end := TOD#00:10:00;
   list[3].shift[3].break[2].end := TOD#02:15:00;
   list[3].shift[3].break[3].end := TOD#03:40:00;
   list[3].shift[3].break[4].end := TOD#04:45:00;
   list[4].shift[0].break[0..4].end := TOD#00:00:00;
   list[4].shift[1].break[0..4].end := TOD#00:00:00;
   list[4].shift[2].break[0..4].end := TOD#00:00:00;
   list[4].shift[3].break[0..4].end := TOD#00:00:00;
   list[5].shift[0].break[0..4].end := TOD#00:00:00;
   list[5].shift[1].break[0..4].end := TOD#00:00:00;
   list[5].shift[2].break[0..4].end := TOD#00:00:00;
   list[5].shift[3].break[0..4].end := TOD#00:00:00;
   list[6].shift[0].break[0..4].end := TOD#00:00:00;
   list[6].shift[1].break[0..4].end := TOD#00:00:00;
   list[6].shift[2].break[0..4].end := TOD#00:00:00;
   list[6].shift[3].break[0..4].end := TOD#00:00:00;
   list[7].shift[0].break[0..4].end := TOD#00:00:00;
   list[7].shift[1].break[0..4].end := TOD#00:00:00;
   list[7].shift[2].break[0..4].end := TOD#00:00:00;
   list[7].shift[3].break[0..4].end := TOD#00:00:00;
   list[8].shift[0].break[0..4].end := TOD#00:00:00;
   list[8].shift[1].break[0..4].end := TOD#00:00:00;
   list[8].shift[2].break[0..4].end := TOD#00:00:00;
   list[8].shift[3].break[0..4].end := TOD#00:00:00;
   list[9].shift[0].break[0..4].end := TOD#00:00:00;
   list[9].shift[1].break[0..4].end := TOD#00:00:00;
   list[9].shift[2].break[0..4].end := TOD#00:00:00;
   list[9].shift[3].break[0..4].end := TOD#00:00:00;
   list[10].shift[0].break[0..4].end := TOD#00:00:00;
   list[10].shift[1].break[0..4].end := TOD#00:00:00;
   list[10].shift[2].break[0..4].end := TOD#00:00:00;
   list[10].shift[3].break[0..4].end := TOD#00:00:00;
   list[0].shift[0..3].end := TOD#00:00:00;
   list[1].shift[0].end := TOD#00:00:00;
   list[1].shift[1].end := TOD#13:30:00;
   list[1].shift[2].end := TOD#21:30:00;
   list[1].shift[3].end := TOD#05:30:00;
   list[2].shift[0].end := TOD#00:00:00;
   list[2].shift[1].end := TOD#14:00:00;
   list[2].shift[2].end := TOD#23:30:00;
   list[2].shift[3].end := TOD#00:00:00;
   list[3].shift[0].end := TOD#00:00:00;
   list[3].shift[1].end := TOD#13:30:00;
   list[3].shift[2].end := TOD#21:30:00;
   list[3].shift[3].end := TOD#05:30:00;
   list[4].shift[0..3].end := TOD#00:00:00;
   list[5].shift[0..3].end := TOD#00:00:00;
   list[6].shift[0..3].end := TOD#00:00:00;
   list[7].shift[0..3].end := TOD#00:00:00;
   list[8].shift[0..3].end := TOD#00:00:00;
   list[9].shift[0..3].end := TOD#00:00:00;
   list[10].shift[0..3].end := TOD#00:00:00;
   list[0].shift[0..3].startCircuitTime := TOD#00:00:00;
   list[1].shift[0].startCircuitTime := TOD#00:00:00;
   list[1].shift[1].startCircuitTime := TOD#13:33:00;
   list[1].shift[2].startCircuitTime := TOD#21:33:00;
   list[1].shift[3].startCircuitTime := TOD#05:33:00;
   list[2].shift[0].startCircuitTime := TOD#00:00:00;
   list[2].shift[1].startCircuitTime := TOD#14:03:00;
   list[2].shift[2].startCircuitTime := TOD#23:33:00;
   list[2].shift[3].startCircuitTime := TOD#00:00:00;
   list[3].shift[0].startCircuitTime := TOD#00:00:00;
   list[3].shift[1].startCircuitTime := TOD#13:33:00;
   list[3].shift[2].startCircuitTime := TOD#21:33:00;
   list[3].shift[3].startCircuitTime := TOD#05:33:00;
   list[4].shift[0..3].startCircuitTime := TOD#00:00:00;
   list[5].shift[0..3].startCircuitTime := TOD#00:00:00;
   list[6].shift[0..3].startCircuitTime := TOD#00:00:00;
   list[7].shift[0..3].startCircuitTime := TOD#00:00:00;
   list[8].shift[0..3].startCircuitTime := TOD#00:00:00;
   list[9].shift[0..3].startCircuitTime := TOD#00:00:00;
   list[10].shift[0..3].startCircuitTime := TOD#00:00:00;
END_DATA_BLOCK

DATA_BLOCK "ManualOperationControl_U1Em0"   // DB104
// stored: MemoryReserve 100
   VAR
      manualOperationEm { ExternalAccessible := 'False'; ExternalVisible := 'False'; ExternalWritable := 'False'} : "LAF_typeManEm";
      manualOperationEmArea { ExternalAccessible := 'False'; ExternalVisible := 'False'; ExternalWritable := 'False'} : Array[1..2] of "LAF_typeManOperationArea";
      manualOperationCms { ExternalAccessible := 'False'; ExternalVisible := 'False'; ExternalWritable := 'False'} : Array[1..90] of "LAF_typeManOperation";
      axis { ExternalAccessible := 'False'; ExternalVisible := 'False'; ExternalWritable := 'False'} : Array[0..0] of "LBC_typeAxisControlInterface";
      axis64Pos { S7_SetPoint := 'True'} : Array[0..20] of "LBC_typeAxis64PosInterface";
      softCam { S7_SetPoint := 'True'} : Array[0..20] of "LER_typeSoftCamInterface2";
      twoWayActuator { S7_SetPoint := 'True'} : Array[0..14] of "LBC_typeTwoWayActuatorInterface";
   END_VAR
BEGIN
   manualOperationEm.equipmentModuleNum := 1010;
   manualOperationEm.actvArea := 0;
   manualOperationEm.pages.total := 0;
   manualOperationEm.pages.actv := 0;
   manualOperationEm.pages.numOfActvItems := 0;
   manualOperationEmArea[1..2].areaNum := 0;
   manualOperationEmArea[1].displayedLines := '1;';
   manualOperationEmArea[2].displayedLines := '21;';
   manualOperationEmArea[1..2].hmiPage.total := 0;
   manualOperationEmArea[1..2].hmiPage.actv := 0;
   manualOperationEmArea[1..2].hmiPage.numOfActvItems := 0;
   manualOperationCms[1..40].intf.lineNum := 0;
   manualOperationCms[1..40].intf.mode := 1;
   manualOperationCms[1..40].intf.showLine := FALSE;
   manualOperationCms[1..40].intf.enableMechAddr := FALSE;
   manualOperationCms[1..40].intf.expandable := FALSE;
   manualOperationCms[1..40].intf.disableLineSel := FALSE;
   manualOperationCms[1..40].intf.enableBigArea := FALSE;
   manualOperationCms[1..40].intf.cnfrmExecLeft := FALSE;
   manualOperationCms[1..40].intf.cnfrmExecRight := FALSE;
   manualOperationCms[1..40].intf.disableLeft := FALSE;
   manualOperationCms[1..40].intf.disableRight := FALSE;
   manualOperationCms[1..40].intf.cnfrmExecLeftCmd := FALSE;
   manualOperationCms[1..40].intf.cnfrmExecRightCmd := FALSE;
   manualOperationCms[1..40].intf.fieldDevAckLeft := FALSE;
   manualOperationCms[1..40].intf.fieldDevAckRight := FALSE;
   manualOperationCms[1..40].intf.nextLeftEndPos := 0;
   manualOperationCms[1..40].intf.nextRightEndPos := 0;
   manualOperationCms[1].intf.leftEndPosSens[0..7] := FALSE;
   manualOperationCms[2].intf.leftEndPosSens[0..7] := FALSE;
   manualOperationCms[3].intf.leftEndPosSens[0..7] := FALSE;
   manualOperationCms[4].intf.leftEndPosSens[0..7] := FALSE;
   manualOperationCms[5].intf.leftEndPosSens[0..7] := FALSE;
   manualOperationCms[6].intf.leftEndPosSens[0..7] := FALSE;
   manualOperationCms[7].intf.leftEndPosSens[0..7] := FALSE;
   manualOperationCms[8].intf.leftEndPosSens[0..7] := FALSE;
   manualOperationCms[9].intf.leftEndPosSens[0..7] := FALSE;
   manualOperationCms[10].intf.leftEndPosSens[0..7] := FALSE;
   manualOperationCms[11].intf.leftEndPosSens[0..7] := FALSE;
   manualOperationCms[12].intf.leftEndPosSens[0..7] := FALSE;
   manualOperationCms[13].intf.leftEndPosSens[0..7] := FALSE;
   manualOperationCms[14].intf.leftEndPosSens[0..7] := FALSE;
   manualOperationCms[15].intf.leftEndPosSens[0..7] := FALSE;
   manualOperationCms[16].intf.leftEndPosSens[0..7] := FALSE;
   manualOperationCms[17].intf.leftEndPosSens[0..7] := FALSE;
   manualOperationCms[18].intf.leftEndPosSens[0..7] := FALSE;
   manualOperationCms[19].intf.leftEndPosSens[0..7] := FALSE;
   manualOperationCms[20].intf.leftEndPosSens[0..7] := FALSE;
   manualOperationCms[21].intf.leftEndPosSens[0..7] := FALSE;
   manualOperationCms[22].intf.leftEndPosSens[0..7] := FALSE;
   manualOperationCms[23].intf.leftEndPosSens[0..7] := FALSE;
   manualOperationCms[24].intf.leftEndPosSens[0..7] := FALSE;
   manualOperationCms[25].intf.leftEndPosSens[0..7] := FALSE;
   manualOperationCms[26].intf.leftEndPosSens[0..7] := FALSE;
   manualOperationCms[27].intf.leftEndPosSens[0..7] := FALSE;
   manualOperationCms[28].intf.leftEndPosSens[0..7] := FALSE;
   manualOperationCms[29].intf.leftEndPosSens[0..7] := FALSE;
   manualOperationCms[30].intf.leftEndPosSens[0..7] := FALSE;
   manualOperationCms[31].intf.leftEndPosSens[0..7] := FALSE;
   manualOperationCms[32].intf.leftEndPosSens[0..7] := FALSE;
   manualOperationCms[33].intf.leftEndPosSens[0..7] := FALSE;
   manualOperationCms[34].intf.leftEndPosSens[0..7] := FALSE;
   manualOperationCms[35].intf.leftEndPosSens[0..7] := FALSE;
   manualOperationCms[36].intf.leftEndPosSens[0..7] := FALSE;
   manualOperationCms[37].intf.leftEndPosSens[0..7] := FALSE;
   manualOperationCms[38].intf.leftEndPosSens[0..7] := FALSE;
   manualOperationCms[39].intf.leftEndPosSens[0..7] := FALSE;
   manualOperationCms[40].intf.leftEndPosSens[0..7] := FALSE;
   manualOperationCms[1].intf.rightEndPosSens[0..7] := FALSE;
   manualOperationCms[2].intf.rightEndPosSens[0..7] := FALSE;
   manualOperationCms[3].intf.rightEndPosSens[0..7] := FALSE;
   manualOperationCms[4].intf.rightEndPosSens[0..7] := FALSE;
   manualOperationCms[5].intf.rightEndPosSens[0..7] := FALSE;
   manualOperationCms[6].intf.rightEndPosSens[0..7] := FALSE;
   manualOperationCms[7].intf.rightEndPosSens[0..7] := FALSE;
   manualOperationCms[8].intf.rightEndPosSens[0..7] := FALSE;
   manualOperationCms[9].intf.rightEndPosSens[0..7] := FALSE;
   manualOperationCms[10].intf.rightEndPosSens[0..7] := FALSE;
   manualOperationCms[11].intf.rightEndPosSens[0..7] := FALSE;
   manualOperationCms[12].intf.rightEndPosSens[0..7] := FALSE;
   manualOperationCms[13].intf.rightEndPosSens[0..7] := FALSE;
   manualOperationCms[14].intf.rightEndPosSens[0..7] := FALSE;
   manualOperationCms[15].intf.rightEndPosSens[0..7] := FALSE;
   manualOperationCms[16].intf.rightEndPosSens[0..7] := FALSE;
   manualOperationCms[17].intf.rightEndPosSens[0..7] := FALSE;
   manualOperationCms[18].intf.rightEndPosSens[0..7] := FALSE;
   manualOperationCms[19].intf.rightEndPosSens[0..7] := FALSE;
   manualOperationCms[20].intf.rightEndPosSens[0..7] := FALSE;
   manualOperationCms[21].intf.rightEndPosSens[0..7] := FALSE;
   manualOperationCms[22].intf.rightEndPosSens[0..7] := FALSE;
   manualOperationCms[23].intf.rightEndPosSens[0..7] := FALSE;
   manualOperationCms[24].intf.rightEndPosSens[0..7] := FALSE;
   manualOperationCms[25].intf.rightEndPosSens[0..7] := FALSE;
   manualOperationCms[26].intf.rightEndPosSens[0..7] := FALSE;
   manualOperationCms[27].intf.rightEndPosSens[0..7] := FALSE;
   manualOperationCms[28].intf.rightEndPosSens[0..7] := FALSE;
   manualOperationCms[29].intf.rightEndPosSens[0..7] := FALSE;
   manualOperationCms[30].intf.rightEndPosSens[0..7] := FALSE;
   manualOperationCms[31].intf.rightEndPosSens[0..7] := FALSE;
   manualOperationCms[32].intf.rightEndPosSens[0..7] := FALSE;
   manualOperationCms[33].intf.rightEndPosSens[0..7] := FALSE;
   manualOperationCms[34].intf.rightEndPosSens[0..7] := FALSE;
   manualOperationCms[35].intf.rightEndPosSens[0..7] := FALSE;
   manualOperationCms[36].intf.rightEndPosSens[0..7] := FALSE;
   manualOperationCms[37].intf.rightEndPosSens[0..7] := FALSE;
   manualOperationCms[38].intf.rightEndPosSens[0..7] := FALSE;
   manualOperationCms[39].intf.rightEndPosSens[0..7] := FALSE;
   manualOperationCms[40].intf.rightEndPosSens[0..7] := FALSE;
   manualOperationCms[1..40].intf.pos := 0.0;
   manualOperationCms[1..40].intf.minPos := 0.0;
   manualOperationCms[1..40].intf.maxPos := 0.0;
   manualOperationCms[1..40].intf.showPos := 0;
   manualOperationCms[1..40].cmd.lineSel := FALSE;
   manualOperationCms[1..40].cmd.expandedOemArea := FALSE;
   manualOperationCms[1..40].cmd.execLeftCmd := FALSE;
   manualOperationCms[1..40].cmd.execRightCmd := FALSE;
   manualOperationCms[1..40].cmd.disableLeftClick := FALSE;
   manualOperationCms[1..40].cmd.disableRightClick := FALSE;
   manualOperationCms[1..40].cmd.moreInfo := FALSE;
   manualOperationCms[1..40].cmd.actvAddr := 1;
   axis[0].commandConfiguration.generalSettings.stopOnError := TRUE;
   axis[0].commandConfiguration.generalSettings.resetWithRestart := FALSE;
   axis[0].commandConfiguration.generalSettings.abortWaitingSyncCmd := TRUE;
   axis[0].commandConfiguration.power.startMode := 1;
   axis[0].commandConfiguration.power.stopMode := 0;
   axis[0].commandConfiguration.power.syncMotionSimulation := FALSE;
   axis[0].commandConfiguration.power.syncMotionSimulationExtendedMode := -1;
   axis[0].commandConfiguration.jog.velocity := 0.0;
   axis[0].commandConfiguration.jog.acceleration := -1.0;
   axis[0].commandConfiguration.jog.deceleration := -1.0;
   axis[0].commandConfiguration.jog.jerk := -1.0;
   axis[0].commandConfiguration.jog.positionControlled := TRUE;
   axis[0].commandConfiguration.jog.increment := 0.0;
   axis[0].commandConfiguration.jog.mode := 0;
   axis[0].commandConfiguration.moveVelocity.velocity := 0.0;
   axis[0].commandConfiguration.moveVelocity.acceleration := -1.0;
   axis[0].commandConfiguration.moveVelocity.deceleration := -1.0;
   axis[0].commandConfiguration.moveVelocity.jerk := -1.0;
   axis[0].commandConfiguration.moveVelocity.direction := 0;
   axis[0].commandConfiguration.moveVelocity.positionControlled := TRUE;
   axis[0].commandConfiguration.moveVelocity.velocityChangeOnTheFly := FALSE;
   axis[0].commandConfiguration.stop.deceleration := -1.0;
   axis[0].commandConfiguration.stop.jerk := -1.0;
   axis[0].commandConfiguration.stop.abortAcceleration := FALSE;
   axis[0].commandConfiguration.fastStop.deceleration := -1.0;
   axis[0].commandConfiguration.fastStop.jerk := -1.0;
   axis[0].commandConfiguration.fastStop.abortAcceleration := FALSE;
   axis[0].commandConfiguration.fastStop.replaceStopPossible := FALSE;
   axis[0].commandConfiguration.torqueLimiting.limit := -1.0;
   axis[0].commandConfiguration.torqueLimiting.mode := 0;
   axis[0].commandConfiguration.homing.position := 0.0;
   axis[0].commandConfiguration.homing.mode := 0;
   axis[0].commandConfiguration.homing.sensor := 0;
   axis[0].commandConfiguration.homing.extendedMode := -1;
   axis[0].commandConfiguration.homing.extendedModeTorqueLimit := 0.0;
   axis[0].commandConfiguration.homing.extendedModeTargetPosition := 0.0;
   axis[0].commandConfiguration.posRelative.distance := 0.0;
   axis[0].commandConfiguration.posRelative.velocity := -1.0;
   axis[0].commandConfiguration.posRelative.acceleration := -1.0;
   axis[0].commandConfiguration.posRelative.deceleration := -1.0;
   axis[0].commandConfiguration.posRelative.jerk := -1.0;
   axis[0].commandConfiguration.posRelative.direction := 0;
   axis[0].commandConfiguration.posAbsolute.position := 0.0;
   axis[0].commandConfiguration.posAbsolute.velocity := -1.0;
   axis[0].commandConfiguration.posAbsolute.acceleration := -1.0;
   axis[0].commandConfiguration.posAbsolute.deceleration := -1.0;
   axis[0].commandConfiguration.posAbsolute.jerk := -1.0;
   axis[0].commandConfiguration.posAbsolute.direction := 1;
   axis[0].commandConfiguration.posAbsolute.positionChangeOnTheFly := FALSE;
   axis[0].commandConfiguration.posAbsolute.velocityChangeOnTheFly := FALSE;
   axis[0].commandConfiguration.posSuperimposed.distance := 0.0;
   axis[0].commandConfiguration.posSuperimposed.velocityDiff := -1.0;
   axis[0].commandConfiguration.posSuperimposed.acceleration := -1.0;
   axis[0].commandConfiguration.posSuperimposed.deceleration := -1.0;
   axis[0].commandConfiguration.posSuperimposed.jerk := -1.0;
   axis[0].commandConfiguration.posSuperimposed.direction := 0;
   axis[0].commandConfiguration.haltSuperimposed.deceleration := -1.0;
   axis[0].commandConfiguration.haltSuperimposed.jerk := -1.0;
   axis[0].commandConfiguration.haltSuperimposed.abortAcceleration := FALSE;
   axis[0].commandConfiguration.gearInRelative.ratioNumerator := 1;
   axis[0].commandConfiguration.gearInRelative.ratioDenominator := 1;
   axis[0].commandConfiguration.gearInRelative.acceleration := -1.0;
   axis[0].commandConfiguration.gearInRelative.deceleration := -1.0;
   axis[0].commandConfiguration.gearInRelative.jerk := -1.0;
   axis[0].commandConfiguration.gearInRelative.ratioChangeOnTheFly := FALSE;
   axis[0].commandConfiguration.gearInAbsolute.ratioNumerator := 1;
   axis[0].commandConfiguration.gearInAbsolute.ratioDenominator := 1;
   axis[0].commandConfiguration.gearInAbsolute.masterSyncPosition := 0.0;
   axis[0].commandConfiguration.gearInAbsolute.slaveSyncPosition := 0.0;
   axis[0].commandConfiguration.gearInAbsolute.syncProfileReference := 1;
   axis[0].commandConfiguration.gearInAbsolute.masterStartDistance := 0.0;
   axis[0].commandConfiguration.gearInAbsolute.velocity := -1.0;
   axis[0].commandConfiguration.gearInAbsolute.acceleration := -1.0;
   axis[0].commandConfiguration.gearInAbsolute.deceleration := -1.0;
   axis[0].commandConfiguration.gearInAbsolute.jerk := -1.0;
   axis[0].commandConfiguration.gearInAbsolute.syncDirection := 1;
   axis[0].commandConfiguration.gearInAbsolute.ratioChangeOnTheFly := FALSE;
   axis[0].commandConfiguration.gearInVelocity.continuousUpdate := FALSE;
   axis[0].commandConfiguration.gearInVelocity.ratioNumerator := 1;
   axis[0].commandConfiguration.gearInVelocity.ratioDenominator := 1;
   axis[0].commandConfiguration.gearInVelocity.acceleration := -1.0;
   axis[0].commandConfiguration.gearInVelocity.deceleration := -1.0;
   axis[0].commandConfiguration.gearInVelocity.jerk := -1.0;
   axis[0].commandConfiguration.gearInVelocity.positionControlled := FALSE;
   axis[0].commandConfiguration.camIn.masterOffset := 0.0;
   axis[0].commandConfiguration.camIn.slaveOffset := 0.0;
   axis[0].commandConfiguration.camIn.masterScaling := 1.0;
   axis[0].commandConfiguration.camIn.slaveScaling := 1.0;
   axis[0].commandConfiguration.camIn.masterSyncPosition := 0.0;
   axis[0].commandConfiguration.camIn.syncProfileReference := 1;
   axis[0].commandConfiguration.camIn.masterStartDistance := 0.0;
   axis[0].commandConfiguration.camIn.velocity := -1.0;
   axis[0].commandConfiguration.camIn.acceleration := -1.0;
   axis[0].commandConfiguration.camIn.deceleration := -1.0;
   axis[0].commandConfiguration.camIn.jerk := -1.0;
   axis[0].commandConfiguration.camIn.applicationMode := 0;
   axis[0].commandConfiguration.camIn.syncDirection := 1;
   axis[0].commandConfiguration.gearOutCamOut.slavePosition := 0.0;
   axis[0].commandConfiguration.gearOutCamOut.syncProfileReference := 1;
   axis[0].commandConfiguration.gearOutCamOut.masterStopDistance := 0.0;
   axis[0].commandConfiguration.gearOutCamOut.deceleration := -1.0;
   axis[0].commandConfiguration.gearOutCamOut.jerk := -1.0;
   axis[0].commandConfiguration.gearOutCamOut.syncOutDirection := 3;
   axis[0].commandConfiguration.gearOutCamOut.gearOutCamOutMode := -1;
   axis[0].commandConfiguration.phasing.phaseShift := 0.0;
   axis[0].commandConfiguration.phasing.velocity := -1.0;
   axis[0].commandConfiguration.phasing.acceleration := -1.0;
   axis[0].commandConfiguration.phasing.deceleration := -1.0;
   axis[0].commandConfiguration.phasing.jerk := -1.0;
   axis[0].commandConfiguration.phasing.profileReference := 0;
   axis[0].commandConfiguration.phasing.phasingDistance := 0.0;
   axis[0].commandConfiguration.phasing.startPosition := 0.0;
   axis[0].commandConfiguration.phasing.direction := 3;
   axis[0].commandConfiguration.phasing.phaseAbsolute := TRUE;
   axis[0].commandConfiguration.phasing.phaseShiftChangeOnTheFly := FALSE;
   axis[0].commandConfiguration.offset.offset := 0.0;
   axis[0].commandConfiguration.offset.profileReference := 1;
   axis[0].commandConfiguration.offset.offsetDistance := 0.0;
   axis[0].commandConfiguration.offset.startPosition := 0.0;
   axis[0].commandConfiguration.offset.direction := 3;
   axis[0].commandConfiguration.offset.offsetAbsolute := TRUE;
   axis[0].commandConfiguration.offset.offsetChangeOnTheFly := FALSE;
   axis[0].commands.enable := FALSE;
   axis[0].commands.enableAxis := FALSE;
   axis[0].commands.resetAxis := FALSE;
   axis[0].commands.openBrake := FALSE;
   axis[0].commands.jogForward := FALSE;
   axis[0].commands.jogBackward := FALSE;
   axis[0].commands.moveVelocity := FALSE;
   axis[0].commands.stop := FALSE;
   axis[0].commands.fastStop := FALSE;
   axis[0].commands.torqueLimiting := FALSE;
   axis[0].commands.homing := FALSE;
   axis[0].commands.posRelative := FALSE;
   axis[0].commands.posAbsolute := FALSE;
   axis[0].commands.posSuperimposed := FALSE;
   axis[0].commands.haltSuperimposed := FALSE;
   axis[0].commands.gearInRelative := FALSE;
   axis[0].commands.gearInAbsolute := FALSE;
   axis[0].commands.gearInVelocity := FALSE;
   axis[0].commands.camIn := FALSE;
   axis[0].commands.gearOutCamOut := FALSE;
   axis[0].commands.phasing := FALSE;
   axis[0].commands.offset := FALSE;
   axis[0].commands.refreshConfiguration := FALSE;
   axis[0].commands.editConfiguration := FALSE;
   axis[0].commands.saveConfiguration := FALSE;
   axis[0].commands.uploadCurrentTorque := FALSE;
   axis[0].commands.reset := FALSE;
   axis[0].monitoring.enable := FALSE;
   axis[0].monitoring.referenceDesignator := WSTRING#'';
   axis[0].monitoring.enabled := FALSE;
   axis[0].monitoring.resetAxis := FALSE;
   axis[0].monitoring.moveVelocity := FALSE;
   axis[0].monitoring.fastStop := FALSE;
   axis[0].monitoring.stop := FALSE;
   axis[0].monitoring.homing := FALSE;
   axis[0].monitoring.posRelative := FALSE;
   axis[0].monitoring.posAbsolute := FALSE;
   axis[0].monitoring.posSuperimposed := FALSE;
   axis[0].monitoring.haltSuperimposed := FALSE;
   axis[0].monitoring.gearInRelative := FALSE;
   axis[0].monitoring.offset := FALSE;
   axis[0].monitoring.phasing := FALSE;
   axis[0].monitoring.gearOutCamOut := FALSE;
   axis[0].monitoring.camIn := FALSE;
   axis[0].monitoring.gearInVelocity := FALSE;
   axis[0].monitoring.gearInAbsolute := FALSE;
   axis[0].monitoring.reset := FALSE;
   axis[0].monitoring.enableAxis := FALSE;
   axis[0].monitoring.openBrake := FALSE;
   axis[0].monitoring.torqueLimiting := FALSE;
   axis[0].monitoring.enableManualCmds := FALSE;
   axis[0].monitoring.jogBackward := FALSE;
   axis[0].monitoring.jogForward := FALSE;
   axis[0].monitoring.brakeOpened := FALSE;
   axis[0].monitoring.axisEnabled := FALSE;
   axis[0].monitoring.resetActive := FALSE;
   axis[0].monitoring.inVelocity := FALSE;
   axis[0].monitoring.inLimitation := FALSE;
   axis[0].monitoring.inClamping := FALSE;
   axis[0].monitoring.startSync := FALSE;
   axis[0].monitoring.inSync := FALSE;
   axis[0].monitoring.inSimulation := FALSE;
   axis[0].monitoring.jogSelected := FALSE;
   axis[0].monitoring.moveVelocitySelected := FALSE;
   axis[0].monitoring.stopSelected := FALSE;
   axis[0].monitoring.fastStopSelected := FALSE;
   axis[0].monitoring.torqueLimitingSelected := FALSE;
   axis[0].monitoring.homingSelected := FALSE;
   axis[0].monitoring.posRelativeSelected := FALSE;
   axis[0].monitoring.posAbsoluteSelected := FALSE;
   axis[0].monitoring.posSuperimposedSelected := FALSE;
   axis[0].monitoring.haltSuperimposedSelected := FALSE;
   axis[0].monitoring.gearInRelativeSelected := FALSE;
   axis[0].monitoring.gearInAbsoluteSelected := FALSE;
   axis[0].monitoring.gearInVelocitySelected := FALSE;
   axis[0].monitoring.camInSelected := FALSE;
   axis[0].monitoring.gearOutCamOutSelected := FALSE;
   axis[0].monitoring.phasingSelected := FALSE;
   axis[0].monitoring.offsetSelected := FALSE;
   axis[0].monitoring.commandBusy := FALSE;
   axis[0].monitoring.commandDone := FALSE;
   axis[0].monitoring.commandAborted := FALSE;
   axis[0].monitoring.homingCommandBusy := FALSE;
   axis[0].monitoring.homingCommandDone := FALSE;
   axis[0].monitoring.homingCommandAborted := FALSE;
   axis[0].monitoring.superimposedBusy := FALSE;
   axis[0].monitoring.superimposedDone := FALSE;
   axis[0].monitoring.superimposedAborted := FALSE;
   axis[0].monitoring.interlockGeneral := FALSE;
   axis[0].monitoring.interlockJogForward := FALSE;
   axis[0].monitoring.interlockJogBackward := FALSE;
   axis[0].monitoring.interlockWarningGeneral := FALSE;
   axis[0].monitoring.interlockWarningJogForward := FALSE;
   axis[0].monitoring.interlockWarningJogBackward := FALSE;
   axis[0].monitoring.valid := FALSE;
   axis[0].monitoring.busy := FALSE;
   axis[0].monitoring.error := FALSE;
   axis[0].monitoring.status := 16#0000;
   axis[0].monitoring.subfunctionStatus := 16#0000;
   axis[0].monitoring.actualPosition := 0.0;
   axis[0].monitoring.actualSpeed := 0.0;
   axis[0].monitoring.speedUnit := 0;
   axis[0].monitoring.positionUnit := 0;
   axis[0].monitoring.axisStatus1 := 16#0000_0000;
   axis[0].monitoring.axisStatus2 := 16#0000_0000;
   axis[0].monitoring.axisType := 0;
   axis[0].monitoring.maxVelocity := 0.0;
   axis[0].monitoring.actualCurrent := 0.0;
   axis[0].monitoring.actualTorque := 0.0;
   axis[0].monitoring.velocityOverrideEnabled := FALSE;
   axis[0].monitoring.sinaParaError := FALSE;
   axis[0].monitoring.sinaParaStatus := 16#0000_0000;
   axis[0].configuration.referenceDesignator := WSTRING#'AxisControl';
   axis[0].configuration.disableAlarms := FALSE;
   axis[0].configuration.masterControlPopUp := TRUE;
   axis64Pos[0..1].commandConfiguration.generalSettings.stopOnError := TRUE;
   axis64Pos[0..1].commandConfiguration.generalSettings.resetWithRestart := FALSE;
   axis64Pos[0..1].commandConfiguration.generalSettings.abortWaitingSyncCmd := TRUE;
   axis64Pos[0..1].commandConfiguration.power.startMode := 1;
   axis64Pos[0..1].commandConfiguration.power.stopMode := 0;
   axis64Pos[0..1].commandConfiguration.power.syncMotionSimulation := FALSE;
   axis64Pos[0..1].commandConfiguration.power.syncMotionSimulationExtendedMode := -1;
   axis64Pos[0..1].commandConfiguration.jog.velocity := 0.0;
   axis64Pos[0..1].commandConfiguration.jog.acceleration := -1.0;
   axis64Pos[0..1].commandConfiguration.jog.deceleration := -1.0;
   axis64Pos[0..1].commandConfiguration.jog.jerk := -1.0;
   axis64Pos[0..1].commandConfiguration.jog.positionControlled := TRUE;
   axis64Pos[0..1].commandConfiguration.jog.increment := 0.0;
   axis64Pos[0..1].commandConfiguration.jog.mode := 0;
   axis64Pos[0..1].commandConfiguration.moveVelocity.velocity := 0.0;
   axis64Pos[0..1].commandConfiguration.moveVelocity.acceleration := -1.0;
   axis64Pos[0..1].commandConfiguration.moveVelocity.deceleration := -1.0;
   axis64Pos[0..1].commandConfiguration.moveVelocity.jerk := -1.0;
   axis64Pos[0..1].commandConfiguration.moveVelocity.direction := 0;
   axis64Pos[0..1].commandConfiguration.moveVelocity.positionControlled := TRUE;
   axis64Pos[0..1].commandConfiguration.moveVelocity.velocityChangeOnTheFly := FALSE;
   axis64Pos[0..1].commandConfiguration.stop.deceleration := -1.0;
   axis64Pos[0..1].commandConfiguration.stop.jerk := -1.0;
   axis64Pos[0..1].commandConfiguration.stop.abortAcceleration := FALSE;
   axis64Pos[0..1].commandConfiguration.fastStop.deceleration := -1.0;
   axis64Pos[0..1].commandConfiguration.fastStop.jerk := -1.0;
   axis64Pos[0..1].commandConfiguration.fastStop.abortAcceleration := FALSE;
   axis64Pos[0..1].commandConfiguration.fastStop.replaceStopPossible := FALSE;
   axis64Pos[0..1].commandConfiguration.torqueLimiting.limit := -1.0;
   axis64Pos[0..1].commandConfiguration.torqueLimiting.mode := 0;
   axis64Pos[0..1].commandConfiguration.homing.position := 0.0;
   axis64Pos[0..1].commandConfiguration.homing.mode := 0;
   axis64Pos[0..1].commandConfiguration.homing.sensor := 0;
   axis64Pos[0..1].commandConfiguration.homing.extendedMode := -1;
   axis64Pos[0..1].commandConfiguration.homing.extendedModeTorqueLimit := 0.0;
   axis64Pos[0..1].commandConfiguration.homing.extendedModeTargetPosition := 0.0;
   axis64Pos[0..1].commandConfiguration.posRelative.distance := 0.0;
   axis64Pos[0..1].commandConfiguration.posRelative.velocity := -1.0;
   axis64Pos[0..1].commandConfiguration.posRelative.acceleration := -1.0;
   axis64Pos[0..1].commandConfiguration.posRelative.deceleration := -1.0;
   axis64Pos[0..1].commandConfiguration.posRelative.jerk := -1.0;
   axis64Pos[0..1].commandConfiguration.posRelative.direction := 0;
   axis64Pos[0..1].commandConfiguration.posAbsolute.position := 0.0;
   axis64Pos[0..1].commandConfiguration.posAbsolute.velocity := -1.0;
   axis64Pos[0..1].commandConfiguration.posAbsolute.acceleration := -1.0;
   axis64Pos[0..1].commandConfiguration.posAbsolute.deceleration := -1.0;
   axis64Pos[0..1].commandConfiguration.posAbsolute.jerk := -1.0;
   axis64Pos[0..1].commandConfiguration.posAbsolute.direction := 1;
   axis64Pos[0..1].commandConfiguration.posAbsolute.positionChangeOnTheFly := FALSE;
   axis64Pos[0..1].commandConfiguration.posAbsolute.velocityChangeOnTheFly := FALSE;
   axis64Pos[0..1].commandConfiguration.posSuperimposed.distance := 0.0;
   axis64Pos[0..1].commandConfiguration.posSuperimposed.velocityDiff := -1.0;
   axis64Pos[0..1].commandConfiguration.posSuperimposed.acceleration := -1.0;
   axis64Pos[0..1].commandConfiguration.posSuperimposed.deceleration := -1.0;
   axis64Pos[0..1].commandConfiguration.posSuperimposed.jerk := -1.0;
   axis64Pos[0..1].commandConfiguration.posSuperimposed.direction := 0;
   axis64Pos[0..1].commandConfiguration.haltSuperimposed.deceleration := -1.0;
   axis64Pos[0..1].commandConfiguration.haltSuperimposed.jerk := -1.0;
   axis64Pos[0..1].commandConfiguration.haltSuperimposed.abortAcceleration := FALSE;
   axis64Pos[0..1].commandConfiguration.gearInRelative.ratioNumerator := 1;
   axis64Pos[0..1].commandConfiguration.gearInRelative.ratioDenominator := 1;
   axis64Pos[0..1].commandConfiguration.gearInRelative.acceleration := -1.0;
   axis64Pos[0..1].commandConfiguration.gearInRelative.deceleration := -1.0;
   axis64Pos[0..1].commandConfiguration.gearInRelative.jerk := -1.0;
   axis64Pos[0..1].commandConfiguration.gearInRelative.ratioChangeOnTheFly := FALSE;
   axis64Pos[0..1].commandConfiguration.gearInAbsolute.ratioNumerator := 1;
   axis64Pos[0..1].commandConfiguration.gearInAbsolute.ratioDenominator := 1;
   axis64Pos[0..1].commandConfiguration.gearInAbsolute.masterSyncPosition := 0.0;
   axis64Pos[0..1].commandConfiguration.gearInAbsolute.slaveSyncPosition := 0.0;
   axis64Pos[0..1].commandConfiguration.gearInAbsolute.syncProfileReference := 1;
   axis64Pos[0..1].commandConfiguration.gearInAbsolute.masterStartDistance := 0.0;
   axis64Pos[0..1].commandConfiguration.gearInAbsolute.velocity := -1.0;
   axis64Pos[0..1].commandConfiguration.gearInAbsolute.acceleration := -1.0;
   axis64Pos[0..1].commandConfiguration.gearInAbsolute.deceleration := -1.0;
   axis64Pos[0..1].commandConfiguration.gearInAbsolute.jerk := -1.0;
   axis64Pos[0..1].commandConfiguration.gearInAbsolute.syncDirection := 1;
   axis64Pos[0..1].commandConfiguration.gearInAbsolute.ratioChangeOnTheFly := FALSE;
   axis64Pos[0..1].commandConfiguration.gearInVelocity.continuousUpdate := FALSE;
   axis64Pos[0..1].commandConfiguration.gearInVelocity.ratioNumerator := 1;
   axis64Pos[0..1].commandConfiguration.gearInVelocity.ratioDenominator := 1;
   axis64Pos[0..1].commandConfiguration.gearInVelocity.acceleration := -1.0;
   axis64Pos[0..1].commandConfiguration.gearInVelocity.deceleration := -1.0;
   axis64Pos[0..1].commandConfiguration.gearInVelocity.jerk := -1.0;
   axis64Pos[0..1].commandConfiguration.gearInVelocity.positionControlled := FALSE;
   axis64Pos[0..1].commandConfiguration.camIn.masterOffset := 0.0;
   axis64Pos[0..1].commandConfiguration.camIn.slaveOffset := 0.0;
   axis64Pos[0..1].commandConfiguration.camIn.masterScaling := 1.0;
   axis64Pos[0..1].commandConfiguration.camIn.slaveScaling := 1.0;
   axis64Pos[0..1].commandConfiguration.camIn.masterSyncPosition := 0.0;
   axis64Pos[0..1].commandConfiguration.camIn.syncProfileReference := 1;
   axis64Pos[0..1].commandConfiguration.camIn.masterStartDistance := 0.0;
   axis64Pos[0..1].commandConfiguration.camIn.velocity := -1.0;
   axis64Pos[0..1].commandConfiguration.camIn.acceleration := -1.0;
   axis64Pos[0..1].commandConfiguration.camIn.deceleration := -1.0;
   axis64Pos[0..1].commandConfiguration.camIn.jerk := -1.0;
   axis64Pos[0..1].commandConfiguration.camIn.applicationMode := 0;
   axis64Pos[0..1].commandConfiguration.camIn.syncDirection := 1;
   axis64Pos[0..1].commandConfiguration.gearOutCamOut.slavePosition := 0.0;
   axis64Pos[0..1].commandConfiguration.gearOutCamOut.syncProfileReference := 1;
   axis64Pos[0..1].commandConfiguration.gearOutCamOut.masterStopDistance := 0.0;
   axis64Pos[0..1].commandConfiguration.gearOutCamOut.deceleration := -1.0;
   axis64Pos[0..1].commandConfiguration.gearOutCamOut.jerk := -1.0;
   axis64Pos[0..1].commandConfiguration.gearOutCamOut.syncOutDirection := 3;
   axis64Pos[0..1].commandConfiguration.gearOutCamOut.gearOutCamOutMode := -1;
   axis64Pos[0..1].commandConfiguration.phasing.phaseShift := 0.0;
   axis64Pos[0..1].commandConfiguration.phasing.velocity := -1.0;
   axis64Pos[0..1].commandConfiguration.phasing.acceleration := -1.0;
   axis64Pos[0..1].commandConfiguration.phasing.deceleration := -1.0;
   axis64Pos[0..1].commandConfiguration.phasing.jerk := -1.0;
   axis64Pos[0..1].commandConfiguration.phasing.profileReference := 0;
   axis64Pos[0..1].commandConfiguration.phasing.phasingDistance := 0.0;
   axis64Pos[0..1].commandConfiguration.phasing.startPosition := 0.0;
   axis64Pos[0..1].commandConfiguration.phasing.direction := 3;
   axis64Pos[0..1].commandConfiguration.phasing.phaseAbsolute := TRUE;
   axis64Pos[0..1].commandConfiguration.phasing.phaseShiftChangeOnTheFly := FALSE;
   axis64Pos[0..1].commandConfiguration.offset.offset := 0.0;
   axis64Pos[0..1].commandConfiguration.offset.profileReference := 1;
   axis64Pos[0..1].commandConfiguration.offset.offsetDistance := 0.0;
   axis64Pos[0..1].commandConfiguration.offset.startPosition := 0.0;
   axis64Pos[0..1].commandConfiguration.offset.direction := 3;
   axis64Pos[0..1].commandConfiguration.offset.offsetAbsolute := TRUE;
   axis64Pos[0..1].commandConfiguration.offset.offsetChangeOnTheFly := FALSE;
   axis64Pos[0..1].commands.enableMasterControl := FALSE;
   axis64Pos[0..1].commands.enableAxis := FALSE;
   axis64Pos[0..1].commands.resetAxis := FALSE;
   axis64Pos[0..1].commands.openBrake := FALSE;
   axis64Pos[0..1].commands.jogForward := FALSE;
   axis64Pos[0..1].commands.jogBackward := FALSE;
   axis64Pos[0..1].commands.moveVelocity := FALSE;
   axis64Pos[0..1].commands.stop := FALSE;
   axis64Pos[0..1].commands.fastStop := FALSE;
   axis64Pos[0..1].commands.torqueLimiting := FALSE;
   axis64Pos[0..1].commands.homing := FALSE;
   axis64Pos[0..1].commands.posRelative := FALSE;
   axis64Pos[0..1].commands.posAbsolute := FALSE;
   axis64Pos[0..1].commands.posSuperimposed := FALSE;
   axis64Pos[0..1].commands.haltSuperimposed := FALSE;
   axis64Pos[0..1].commands.selectSetPosition := 0;
   axis64Pos[0..1].commands.uploadParameters := FALSE;
   axis64Pos[0..1].commands.refreshConfiguration := FALSE;
   axis64Pos[0..1].commands.editConfiguration := FALSE;
   axis64Pos[0..1].commands.saveConfiguration := FALSE;
   axis64Pos[0..1].commands.uploadCurrentTorque := FALSE;
   axis64Pos[0..1].commands.reset := FALSE;
   axis64Pos[0..1].monitoring.enable := FALSE;
   axis64Pos[0..1].monitoring.referenceDesignator := WSTRING#'';
   axis64Pos[0..1].monitoring.enabled := FALSE;
   axis64Pos[0..1].monitoring.enableManualCmds := FALSE;
   axis64Pos[0..1].monitoring.reset := FALSE;
   axis64Pos[0..1].monitoring.resetAxis := FALSE;
   axis64Pos[0..1].monitoring.enableAxis := FALSE;
   axis64Pos[0..1].monitoring.openBrake := FALSE;
   axis64Pos[0..1].monitoring.jogBackward := FALSE;
   axis64Pos[0..1].monitoring.jogForward := FALSE;
   axis64Pos[0..1].monitoring.moveVelocity := FALSE;
   axis64Pos[0..1].monitoring.stop := FALSE;
   axis64Pos[0..1].monitoring.fastStop := FALSE;
   axis64Pos[0..1].monitoring.torqueLimiting := FALSE;
   axis64Pos[0..1].monitoring.homing := FALSE;
   axis64Pos[0..1].monitoring.posRelative := FALSE;
   axis64Pos[0..1].monitoring.posAbsolute := FALSE;
   axis64Pos[0..1].monitoring.posSuperimposed := FALSE;
   axis64Pos[0..1].monitoring.haltSuperimposed := FALSE;
   axis64Pos[0..1].monitoring.brakeOpened := FALSE;
   axis64Pos[0..1].monitoring.axisEnabled := FALSE;
   axis64Pos[0..1].monitoring.resetActive := FALSE;
   axis64Pos[0..1].monitoring.inVelocity := FALSE;
   axis64Pos[0..1].monitoring.inLimitation := FALSE;
   axis64Pos[0..1].monitoring.inClamping := FALSE;
   axis64Pos[0..1].monitoring.startSync := FALSE;
   axis64Pos[0..1].monitoring.inSync := FALSE;
   axis64Pos[0..1].monitoring.inSimulation := FALSE;
   axis64Pos[0..1].monitoring.jogSelected := FALSE;
   axis64Pos[0..1].monitoring.moveVelocitySelected := FALSE;
   axis64Pos[0..1].monitoring.stopSelected := FALSE;
   axis64Pos[0..1].monitoring.fastStopSelected := FALSE;
   axis64Pos[0..1].monitoring.torqueLimitingSelected := FALSE;
   axis64Pos[0..1].monitoring.homingSelected := FALSE;
   axis64Pos[0..1].monitoring.posRelativeSelected := FALSE;
   axis64Pos[0..1].monitoring.posAbsoluteSelected := FALSE;
   axis64Pos[0..1].monitoring.posSuperimposedSelected := FALSE;
   axis64Pos[0..1].monitoring.haltSuperimposedSelected := FALSE;
   axis64Pos[0..1].monitoring.commandBusy := FALSE;
   axis64Pos[0..1].monitoring.commandDone := FALSE;
   axis64Pos[0..1].monitoring.commandAborted := FALSE;
   axis64Pos[0..1].monitoring.homingCommandBusy := FALSE;
   axis64Pos[0..1].monitoring.homingCommandDone := FALSE;
   axis64Pos[0..1].monitoring.homingCommandAborted := FALSE;
   axis64Pos[0..1].monitoring.superimposedBusy := FALSE;
   axis64Pos[0..1].monitoring.superimposedDone := FALSE;
   axis64Pos[0..1].monitoring.superimposedAborted := FALSE;
   axis64Pos[0..1].monitoring.selectSetPosition := 0;
   axis64Pos[0..1].monitoring.selectionController := TRUE;
   axis64Pos[0..1].monitoring.interlockGeneral := FALSE;
   axis64Pos[0..1].monitoring.interlockJogForward := FALSE;
   axis64Pos[0..1].monitoring.interlockJogBackward := FALSE;
   axis64Pos[0..1].monitoring.interlockWarningGeneral := FALSE;
   axis64Pos[0..1].monitoring.interlockWarningJogForward := FALSE;
   axis64Pos[0..1].monitoring.interlockWarningJogBackward := FALSE;
   axis64Pos[0..1].monitoring.valid := FALSE;
   axis64Pos[0..1].monitoring.busy := FALSE;
   axis64Pos[0..1].monitoring.error := FALSE;
   axis64Pos[0..1].monitoring.status := 16#0000;
   axis64Pos[0..1].monitoring.subfunctionStatus := 16#0000;
   axis64Pos[0..1].monitoring.actualPosition := 0.0;
   axis64Pos[0..1].monitoring.actualSpeed := 0.0;
   axis64Pos[0..1].monitoring.speedUnit := 0;
   axis64Pos[0..1].monitoring.positionUnit := 0;
   axis64Pos[0..1].monitoring.axisType := 0;
   axis64Pos[0..1].monitoring.maxVelocity := 0.0;
   axis64Pos[0..1].monitoring.actualCurrent := 0.0;
   axis64Pos[0..1].monitoring.actualTorque := 0.0;
   axis64Pos[0..1].monitoring.velocityOverrideEnabled := FALSE;
   axis64Pos[0..1].monitoring.sinaParaError := FALSE;
   axis64Pos[0..1].monitoring.sinaParaStatus := 16#0000_0000;
   axis64Pos[0..1].configuration.referenceDesignator := WSTRING#'Axis64Pos';
   axis64Pos[0..1].configuration.disableAlarms := FALSE;
   axis64Pos[0..1].configuration.masterControlPopUp := TRUE;
   axis64Pos[0].configuration.setPositions[0..15].position := 0.0;
   axis64Pos[1].configuration.setPositions[0..15].position := 0.0;
   axis64Pos[0].configuration.setPositions[0..15].velocity := -1.0;
   axis64Pos[1].configuration.setPositions[0..15].velocity := -1.0;
   axis64Pos[0].configuration.setPositions[0..15].acceleration := -1.0;
   axis64Pos[1].configuration.setPositions[0..15].acceleration := -1.0;
   axis64Pos[0].configuration.setPositions[0..15].deceleration := -1.0;
   axis64Pos[1].configuration.setPositions[0..15].deceleration := -1.0;
   axis64Pos[0].configuration.setPositions[0..15]."name" := '';
   axis64Pos[1].configuration.setPositions[0..15]."name" := '';
   twoWayActuator[0..1].commands.refreshConfiguration := FALSE;
   twoWayActuator[0..1].commands.editConfiguration := FALSE;
   twoWayActuator[0..1].commands.saveConfiguration := FALSE;
   twoWayActuator[0..1].commands.reset := FALSE;
   twoWayActuator[0..1].commands.commandHomePos := FALSE;
   twoWayActuator[0..1].commands.commandWorkPos := FALSE;
   twoWayActuator[0..1].monitoring.enable := FALSE;
   twoWayActuator[0..1].monitoring.referenceDesignator := WSTRING#'';
   twoWayActuator[0..1].monitoring.commandHomePos := FALSE;
   twoWayActuator[0..1].monitoring.commandWorkPos := FALSE;
   twoWayActuator[0..1].monitoring.goToHomePos := FALSE;
   twoWayActuator[0..1].monitoring.goToWorkPos := FALSE;
   twoWayActuator[0..1].monitoring.inHomePos := FALSE;
   twoWayActuator[0..1].monitoring.inWorkPos := FALSE;
   twoWayActuator[0..1].monitoring.reset := FALSE;
   twoWayActuator[0..1].monitoring.enableManualCmds := FALSE;
   twoWayActuator[0..1].monitoring.error := FALSE;
   twoWayActuator[0..1].monitoring.interlockHomePos := FALSE;
   twoWayActuator[0..1].monitoring.interlockWorkPos := FALSE;
   twoWayActuator[0..1].monitoring.status := 16#0000;
   twoWayActuator[0..1].monitoring.interlockWarningWorkPos := FALSE;
   twoWayActuator[0..1].monitoring.interlockWarningHomePos := FALSE;
   twoWayActuator[0..1].configuration.referenceDesignator := WSTRING#'TwoWayAct.';
   twoWayActuator[0..1].configuration.monitoringLeavingFeedback := T#5S;
   twoWayActuator[0..1].configuration.monitoringReachingFeedback := T#5S;
   twoWayActuator[0..1].configuration.monitoringDiscrepancy := T#0MS;
   twoWayActuator[0..1].configuration.setOutputHomeContinuously := TRUE;
   twoWayActuator[0..1].configuration.setOutputWorkContinuously := TRUE;
   twoWayActuator[0..1].configuration.disableHomeCommand := FALSE;
   twoWayActuator[0..1].configuration.disableFeedbackHomePos := FALSE;
   twoWayActuator[0..1].configuration.disableFeedbackWorkPos := FALSE;
   twoWayActuator[0..1].configuration.disableAlarms := FALSE;
   twoWayActuator[0..1].configuration.resetOutputsOnError := FALSE;
   twoWayActuator[0..1].configuration.allwaysWaitOnReachingTime := FALSE;
END_DATA_BLOCK

DATA_BLOCK "DriveDiagInterfaceHmi"   // DB46
TITLE = DriveDiagInterfaceHmi
AUTHOR : Siemens Digital Industries
FAMILY : LAF
NAME : LAF_DriveDiagInterfaceHmi
VERSION : 1.1
// HMI interface for drive diagnostic
// stored: MemoryReserve 100
   VAR
      diagStatus : "LAF_typeDriveDiagInterfaceHmi";
   END_VAR
BEGIN
   diagStatus.hmi.referenceDesignator := WSTRING#'';
   diagStatus.hmi.driveIndex := 0;
   diagStatus.hmi.axisStatusScreenActive := FALSE;
   diagStatus.hmi.sinaStatusScreenActive := FALSE;
   diagStatus.hmi.sinaAlarmScreenActive := FALSE;
   diagStatus.hmi.sinaEposScreenActive := FALSE;
   diagStatus.hmi.sinaSafetyScreenActive := FALSE;
   diagStatus.axis."type" := 0;
   diagStatus.axis.values.position := 0.0;
   diagStatus.axis.values.velocity := 0.0;
   diagStatus.axis.values.actualPosition := 0.0;
   diagStatus.axis.values.actualVelocity := 0.0;
   diagStatus.axis.values.actualSpeed := 0.0;
   diagStatus.axis.statusAxis.statusWord := 16#0000_0000;
   diagStatus.axis.statusAxis.statusWord2 := 16#0000_0000;
   diagStatus.axis.statusAxis.warningWord := 16#0000_0000;
   diagStatus.axis.statusAxis.errorWord := 16#0000_0000;
   diagStatus.axis.statusAxis.status.bit00_Enable := FALSE;
   diagStatus.axis.statusAxis.status.bit01_Error := FALSE;
   diagStatus.axis.statusAxis.status.bit02_RestartActive := FALSE;
   diagStatus.axis.statusAxis.status.bit03_OnlineStartValuesChanged := FALSE;
   diagStatus.axis.statusAxis.status.bit04_ControlPanelActive := FALSE;
   diagStatus.axis.statusAxis.status.bit05_HomingDone := FALSE;
   diagStatus.axis.statusAxis.status.bit06_Done := FALSE;
   diagStatus.axis.statusAxis.status.bit07_Standstill := FALSE;
   diagStatus.axis.statusAxis.status.bit08_PositioningCommand := FALSE;
   diagStatus.axis.statusAxis.status.bit09_JogCommand := FALSE;
   diagStatus.axis.statusAxis.status.bit10_VelocityCommand := FALSE;
   diagStatus.axis.statusAxis.status.bit11_HomingCommand := FALSE;
   diagStatus.axis.statusAxis.status.bit12_ConstantVelocity := FALSE;
   diagStatus.axis.statusAxis.status.bit13_Accelerating := FALSE;
   diagStatus.axis.statusAxis.status.bit14_Decelerating := FALSE;
   diagStatus.axis.statusAxis.status.bit15_SWLimitMinActive := FALSE;
   diagStatus.axis.statusAxis.status.bit16_SWLimitMaxActive := FALSE;
   diagStatus.axis.statusAxis.status.bit17_HWLimitMinActive := FALSE;
   diagStatus.axis.statusAxis.status.bit18_HWLimitMaxActive := FALSE;
   diagStatus.axis.statusAxis.status.bit19_Reserved := FALSE;
   diagStatus.axis.statusAxis.status.bit20_Reserved := FALSE;
   diagStatus.axis.statusAxis.status.bit21_Synchronizing := FALSE;
   diagStatus.axis.statusAxis.status.bit22_Synchronous := FALSE;
   diagStatus.axis.statusAxis.status.bit23_SuperimposedMotionCommand := FALSE;
   diagStatus.axis.statusAxis.status.bit24_PhasingCommand := FALSE;
   diagStatus.axis.statusAxis.status.bit25_AxisSimulation := FALSE;
   diagStatus.axis.statusAxis.status.bit26_TorqueLimitingCommand := FALSE;
   diagStatus.axis.statusAxis.status.bit27_InLimitation := FALSE;
   diagStatus.axis.statusAxis.status.bit28_NonPositionControlled := FALSE;
   diagStatus.axis.statusAxis.status.bit29_KinematicsMotionCommand := FALSE;
   diagStatus.axis.statusAxis.status.bit30_InClamping := FALSE;
   diagStatus.axis.statusAxis.status.bit31_MotionInCommand := FALSE;
   diagStatus.axis.statusAxis.status2.bit00_StopCommand := FALSE;
   diagStatus.axis.statusAxis.status2.bit01_DesynchronizingCommand := FALSE;
   diagStatus.axis.statusAxis.status2.bit02_PassingBacklash := FALSE;
   diagStatus.axis.statusAxis.status2.bit03_PhasingCommandWaiting := FALSE;
   diagStatus.axis.statusAxis.status2.bit04_OffsetCommand := FALSE;
   diagStatus.axis.statusAxis.status2.bit05_OffsetCommandWaiting := FALSE;
   diagStatus.axis.statusAxis.status2.bit06_MotionInSuperimposedCommand := FALSE;
   diagStatus.axis.statusAxis.status2.bit07_HaltSuperimposedCommand := FALSE;
   diagStatus.axis.statusAxis.status2.bit08_Reserved := FALSE;
   diagStatus.axis.statusAxis.status2.bit09_Reserved := FALSE;
   diagStatus.axis.statusAxis.status2.bit10_Reserved := FALSE;
   diagStatus.axis.statusAxis.status2.bit11_Reserved := FALSE;
   diagStatus.axis.statusAxis.status2.bit12_Reserved := FALSE;
   diagStatus.axis.statusAxis.status2.bit13_Reserved := FALSE;
   diagStatus.axis.statusAxis.status2.bit14_Reserved := FALSE;
   diagStatus.axis.statusAxis.status2.bit15_Reserved := FALSE;
   diagStatus.axis.statusAxis.status2.bit16_Reserved := FALSE;
   diagStatus.axis.statusAxis.status2.bit17_Reserved := FALSE;
   diagStatus.axis.statusAxis.status2.bit18_Reserved := FALSE;
   diagStatus.axis.statusAxis.status2.bit19_Reserved := FALSE;
   diagStatus.axis.statusAxis.status2.bit20_Reserved := FALSE;
   diagStatus.axis.statusAxis.status2.bit21_Reserved := FALSE;
   diagStatus.axis.statusAxis.status2.bit22_Reserved := FALSE;
   diagStatus.axis.statusAxis.status2.bit23_Reserved := FALSE;
   diagStatus.axis.statusAxis.status2.bit24_Reserved := FALSE;
   diagStatus.axis.statusAxis.status2.bit25_Reserved := FALSE;
   diagStatus.axis.statusAxis.status2.bit26_Reserved := FALSE;
   diagStatus.axis.statusAxis.status2.bit27_Reserved := FALSE;
   diagStatus.axis.statusAxis.status2.bit28_Reserved := FALSE;
   diagStatus.axis.statusAxis.status2.bit29_Reserved := FALSE;
   diagStatus.axis.statusAxis.status2.bit30_Reserved := FALSE;
   diagStatus.axis.statusAxis.status2.bit31_Reserved := FALSE;
   diagStatus.axis.statusAxis.warning.bit00_SystemWarning := FALSE;
   diagStatus.axis.statusAxis.warning.bit01_ConfigWarning := FALSE;
   diagStatus.axis.statusAxis.warning.bit02_UserWarning := FALSE;
   diagStatus.axis.statusAxis.warning.bit03_CommandNotAccepted := FALSE;
   diagStatus.axis.statusAxis.warning.bit04_DriveWarning := FALSE;
   diagStatus.axis.statusAxis.warning.bit05_SensorWarning := FALSE;
   diagStatus.axis.statusAxis.warning.bit06_DynamicWarning := FALSE;
   diagStatus.axis.statusAxis.warning.bit07_CommunicationWarning := FALSE;
   diagStatus.axis.statusAxis.warning.bit08_SWLimitMin := FALSE;
   diagStatus.axis.statusAxis.warning.bit09_SWLimitMax := FALSE;
   diagStatus.axis.statusAxis.warning.bit10_HomingWarning := FALSE;
   diagStatus.axis.statusAxis.warning.bit11_FollowingErrorWarning := FALSE;
   diagStatus.axis.statusAxis.warning.bit12_PositioningWarning := FALSE;
   diagStatus.axis.statusAxis.warning.bit13_PeripheralWarning := FALSE;
   diagStatus.axis.statusAxis.warning.bit14_SynchronousWarning := FALSE;
   diagStatus.axis.statusAxis.warning.bit15_AdaptionWarning := FALSE;
   diagStatus.axis.statusAxis.warning.bit16_Reserved := FALSE;
   diagStatus.axis.statusAxis.warning.bit17_Reserved := FALSE;
   diagStatus.axis.statusAxis.warning.bit18_Reserved := FALSE;
   diagStatus.axis.statusAxis.warning.bit19_Reserved := FALSE;
   diagStatus.axis.statusAxis.warning.bit20_Reserved := FALSE;
   diagStatus.axis.statusAxis.warning.bit21_Reserved := FALSE;
   diagStatus.axis.statusAxis.warning.bit22_Reserved := FALSE;
   diagStatus.axis.statusAxis.warning.bit23_Reserved := FALSE;
   diagStatus.axis.statusAxis.warning.bit24_Reserved := FALSE;
   diagStatus.axis.statusAxis.warning.bit25_Reserved := FALSE;
   diagStatus.axis.statusAxis.warning.bit26_Reserved := FALSE;
   diagStatus.axis.statusAxis.warning.bit27_Reserved := FALSE;
   diagStatus.axis.statusAxis.warning.bit28_Reserved := FALSE;
   diagStatus.axis.statusAxis.warning.bit29_Reserved := FALSE;
   diagStatus.axis.statusAxis.warning.bit30_Reserved := FALSE;
   diagStatus.axis.statusAxis.warning.bit31_Reserved := FALSE;
   diagStatus.axis.statusAxis.error.bit00_SystemFault := FALSE;
   diagStatus.axis.statusAxis.error.bit01_ConfigFault := FALSE;
   diagStatus.axis.statusAxis.error.bit02_UserFault := FALSE;
   diagStatus.axis.statusAxis.error.bit03_CommandNotAccepted := FALSE;
   diagStatus.axis.statusAxis.error.bit04_DriveFault := FALSE;
   diagStatus.axis.statusAxis.error.bit05_SensorFault := FALSE;
   diagStatus.axis.statusAxis.error.bit06_DynamicError := FALSE;
   diagStatus.axis.statusAxis.error.bit07_CommunicationFault := FALSE;
   diagStatus.axis.statusAxis.error.bit08_SWLimit := FALSE;
   diagStatus.axis.statusAxis.error.bit09_HWLimit := FALSE;
   diagStatus.axis.statusAxis.error.bit10_HomingError := FALSE;
   diagStatus.axis.statusAxis.error.bit11_FollowingErrorFault := FALSE;
   diagStatus.axis.statusAxis.error.bit12_PositioningFault := FALSE;
   diagStatus.axis.statusAxis.error.bit13_PeripheralError := FALSE;
   diagStatus.axis.statusAxis.error.bit14_SynchronousError := FALSE;
   diagStatus.axis.statusAxis.error.bit15_AdaptionError := FALSE;
   diagStatus.axis.statusAxis.error.bit16_Reserved := FALSE;
   diagStatus.axis.statusAxis.error.bit17_Reserved := FALSE;
   diagStatus.axis.statusAxis.error.bit18_Reserved := FALSE;
   diagStatus.axis.statusAxis.error.bit19_Reserved := FALSE;
   diagStatus.axis.statusAxis.error.bit20_Reserved := FALSE;
   diagStatus.axis.statusAxis.error.bit21_Reserved := FALSE;
   diagStatus.axis.statusAxis.error.bit22_Reserved := FALSE;
   diagStatus.axis.statusAxis.error.bit23_Reserved := FALSE;
   diagStatus.axis.statusAxis.error.bit24_Reserved := FALSE;
   diagStatus.axis.statusAxis.error.bit25_Reserved := FALSE;
   diagStatus.axis.statusAxis.error.bit26_Reserved := FALSE;
   diagStatus.axis.statusAxis.error.bit27_Reserved := FALSE;
   diagStatus.axis.statusAxis.error.bit28_Reserved := FALSE;
   diagStatus.axis.statusAxis.error.bit29_Reserved := FALSE;
   diagStatus.axis.statusAxis.error.bit30_Reserved := FALSE;
   diagStatus.axis.statusAxis.error.bit31_Reserved := FALSE;
   diagStatus.axis.statusAxis.errorDetail.number := 0;
   diagStatus.axis.statusAxis.errorDetail.reaction := 0;
   diagStatus.axis.statusSensor.operativeSensor := 1;
   diagStatus.axis.statusSensor.sensor[1..4].state := 0;
   diagStatus.axis.statusSensor.sensor[1..4].communicationOK := FALSE;
   diagStatus.axis.statusSensor.sensor[1..4].error := FALSE;
   diagStatus.axis.statusSensor.sensor[1..4].control := FALSE;
   diagStatus.axis.statusSensor.sensor[1..4].position := 0.0;
   diagStatus.axis.statusSensor.sensor[1..4].velocity := 0.0;
   diagStatus.axis.statusSensor.sensor[1..4].adaptionState := 0;
   diagStatus.axis.statusSensor.sensor[1..4].adjusted := 0;
   diagStatus.axis.statusPositioning.targetPosition := 0.0;
   diagStatus.axis.statusPositioning.followingError := 0.0;
   diagStatus.axis.units.lengthUnit := 0;
   diagStatus.axis.units.velocityUnit := 0;
   diagStatus.sina.sinaType := 0;
   diagStatus.sina.controlWord := 16#0000;
   diagStatus.sina.statusWord := 16#0000;
   diagStatus.sina.telegramNo := 0;
   diagStatus.sina.eposStatusWord1 := 16#0000;
   diagStatus.sina.eposStatusWord2 := 16#0000;
   diagStatus.sina.operatingDisplay := 0;
   diagStatus.sina.override := 0.0;
   diagStatus.sina.posSetValue := 0.0;
   diagStatus.sina.posActValue := 0.0;
   diagStatus.sina.velSetValue := 0.0;
   diagStatus.sina.velActValue := 0.0;
   diagStatus.sina.lengthUnit := 0;
   diagStatus.sina.velocityUnit := 0;
   diagStatus.sina.residualDistance := 0.0;
   diagStatus.sina.followingError := 0.0;
   diagStatus.sina.posControlWord := 16#0000;
   diagStatus.sina.posStatusWord := 16#0000;
   diagStatus.sina.blockSelected := 0;
   diagStatus.sina.blockActive := 0;
   diagStatus.sina.mdiPosSetValue := 0.0;
   diagStatus.sina.faultCode[0..7] := 16#0000;
   diagStatus.sina.alarmCode[0..3] := 16#0000;
   diagStatus.sina.speedSetValue := 0.0;
   diagStatus.sina.speedActValue := 0.0;
   diagStatus.sina.safetyStatusWord := 16#0000;
END_DATA_BLOCK

DATA_BLOCK "TestVarIdent"   // DB76
TITLE = Test tags fuer ident / Test tags for ident
AUTHOR : SICAR
FAMILY : Ident
VERSION : 1.0
// Test tags fuer ident / Test tags for ident
// stored: MemoryReserve 100
   VAR
      init1 : Bool := FALSE;   // Init 1
      read1 : Bool := FALSE;   // Read1
      write1 : Bool := FALSE;   // Write1
      init2 : Bool := FALSE;   // Init 2
      read2 : Bool := FALSE;   // Read2
      write2 : Bool := FALSE;   // Write2
      testString : String[32] := '';   // Test string
      charArr : Array[1..32] of Byte;   // Array of characters / Character Array
      prgNoMan : USInt := 0;   // Progrmm Nummer schreiben manual / Program number manual
      enableManCtrlRf : Bool := FALSE;   // Freigabe Manual Steuerung / Enable manual control RFID
      enableOption : Bool := FALSE;   // Freiegbae Optionen / Enable options
      enableManCtrlMV : Bool := FALSE;   // Enable manual control MV
   END_VAR
BEGIN
   charArr[1..32] := 16#00;
END_DATA_BLOCK

DATA_BLOCK "PM02"   // DB336
// stored: MemoryReserve 100
   VAR
      "SUCTION PAD #1 TOP UP" : Bool := FALSE;
      "SUCTION PAD #1 TOP DOWN" : Bool := FALSE;
      "SUCTION PAD #1 BTM UP" : Bool := FALSE;
      "SUCTION PAD #1 BTM DOWN" : Bool := FALSE;
      "CUTTER #1 UP" : Bool := FALSE;
      "CUTTER #1 DOWN" : Bool := FALSE;
      "TAPE #1 TOP UP" : Bool := FALSE;
      "TAPE #1 TOP DOWN" : Bool := FALSE;
      "TAPE #1 BTM UP" : Bool := FALSE;
      "TAPE #1 BTM DOWN" : Bool := FALSE;
      "SPLICE HEAD ROTATE #1 TOP FORWARD" : Bool := FALSE;
      "SPLICE HEAD ROTATE #1 TOP BACKWARD" : Bool := FALSE;
      "SPLICE HEAD ROTATE #1 BTM FORWARD" : Bool := FALSE;
      "SPLICE HEAD ROTATE #1 BTM BACKWARD" : Bool := FALSE;
   END_VAR
BEGIN
END_DATA_BLOCK

DATA_BLOCK "PM06"   // DB335
// stored: MemoryReserve 100
   VAR
      "CATHODE GLASS CLEANING ON" : Bool := FALSE;
      SPARE : Bool := FALSE;
      "CATHODE MAIN NG P&P UP" : Bool := FALSE;
      "CATHODE MAIN NG P&P DOWN" : Bool := FALSE;
      "CATHODE MAIN NG P&P 1st FORWARD" : Bool := FALSE;
      "CATHODE MAIN NG P&P 1st BACKWARD" : Bool := FALSE;
      "CATHODE MAIN NG P&P 2nd FORWARD" : Bool := FALSE;
      "CATHODE MAIN NG P&P 2nd BACKWARD" : Bool := FALSE;
      "CATHODE FIX FRONT&REAR FORWARD" : Bool := FALSE;
      "CATHODE FIX FRONT&REAR BACKWARD" : Bool := FALSE;
      "CATHODE MAIN P&P#1 Rotary CW" : Bool := FALSE;
      "CATHODE MAIN P&P#1 Rotary CCW" : Bool := FALSE;
      "CATHODE NG BOX LIFT UP" : Bool := FALSE;
      "CATHODE NG BOX LIFT DOWN" : Bool := FALSE;
      "CATHODE NG BOX LOCK UP" : Bool := FALSE;
      "CATHODE NG BOX LOCK DOWN" : Bool := FALSE;
   END_VAR
BEGIN
END_DATA_BLOCK

DATA_BLOCK "SBK01"   // DB322
// stored: MemoryReserve 100
   VAR
      SPARE : Bool := FALSE;
      "EMO02 CH.A" : Bool := TRUE;
      SPARE_1 : Bool := FALSE;
      "EMO04 CH.A" : Bool := TRUE;
      "EMO01 CH.B" : Bool;
      "EMO02 CH.B" : Bool;
      SPARE_2 : Bool;
      "EMO04 CH.B" : Bool;
      SPARE_3 : Bool;
      SPARE_4 : Bool;
      SPARE_5 : Bool;
   END_VAR
BEGIN
END_DATA_BLOCK

DATA_BLOCK "SBK07"   // DB320
// stored: MemoryReserve 100
   VAR
      "GATE EC SCRAP BOX-1 PB.LOCK" : Bool := FALSE;
      "GATE EC SCRAP BOX-1 PB.RESET" : Bool := FALSE;
      SPARE : Bool := FALSE;
      SPARE_1 : Bool := FALSE;
      "GATE EC SCRAP BOX-1 PB.UNLOCK" : Bool := FALSE;
      SPARE_2 : Bool := FALSE;
      SPARE_3 : Bool := FALSE;
      SPARE_4 : Bool := FALSE;
      "GATE EC SCRAP BOX-1 PL.LOCK" : Bool := FALSE;
      "GATE EC SCRAP BOX-1 PL.UNLOCK" : Bool := TRUE;
      "GATE EC SCRAP BOX-1 PL.RESET" : Bool := FALSE;
   END_VAR
BEGIN
END_DATA_BLOCK

DATA_BLOCK "SBK08"   // DB321
// stored: MemoryReserve 100
   VAR
      "SAFETY DOOR LOCK1.INPUT" : Bool := TRUE;
      "SAFETY DOOR LOCK2.INPUT" : Bool := TRUE;
      "SAFETY DOOR LOCK3.INPUT" : Bool := TRUE;
      SPARE : Bool := FALSE;
      "SAFETY DOOR LOCK1.INPUT_1" : Bool := FALSE;
      "SAFETY DOOR LOCK2.INPUT_1" : Bool := FALSE;
      "SAFETY DOOR LOCK3.INPUT_1" : Bool := FALSE;
      SPARE_1 : Bool := FALSE;
      "SAFETY DOOR LOCK1.OUTPUT" : Bool := FALSE;
      "SAFETY DOOR LOCK2.OUTPUT" : Bool := FALSE;
      "SAFETY DOOR LOCK3.OUTPUT" : Bool := FALSE;
   END_VAR
BEGIN
END_DATA_BLOCK

DATA_BLOCK "SBK09"   // DB326
// stored: MemoryReserve 100
   VAR
      "SAFETY DOOR LOCK4.INPUT" : Bool := TRUE;
      "SAFETY DOOR LOCK5.INPUT" : Bool := TRUE;
      SPARE_5 : Bool := TRUE;
      SPARE : Bool := FALSE;
      "SAFETY DOOR LOCK4.INPUT_1" : Bool := FALSE;
      "SAFETY DOOR LOCK5.INPUT_1" : Bool := FALSE;
      SPARE_2 : Bool := FALSE;
      SPARE_3 : Bool := FALSE;
      "SAFETY DOOR LOCK4.OUTPUT" : Bool := FALSE;
      "SAFETY DOOR LOCK5.OUTPUT" : Bool := FALSE;
      SPARE_4 : Bool := FALSE;
   END_VAR
BEGIN
END_DATA_BLOCK

DATA_BLOCK "SP203"   // DB346
// stored: MemoryReserve 100
   VAR
      "MAIN OP MODE SLELECT SS.AUTO" : Bool := FALSE;
      "MAIN OP HOME PBL (GREEN)" : Bool := FALSE;
      "MAIN OP SAFETY RESET PBL (BLUE)" : Bool := FALSE;
      "MAIN OP SCS MODE SLELECT SS.AUTO" : Bool := FALSE;
      "MAIN OP MODE SLELECT SS.MANUAL" : Bool := TRUE;
      "MAIN OP ENABLE PBL (WHITE)" : Bool := FALSE;
      "MAIN OP SCS MODE SLELECT SS.SETUP" : Bool := TRUE;
      "MAIN OP SCS MODE SLELECT SS.DISABLE" : Bool := FALSE;
   END_VAR
BEGIN
END_DATA_BLOCK

DATA_BLOCK "SP502"   // DB349
// stored: MemoryReserve 100
   VAR
      "CLASS2 SMPS ALARM RESET" : Bool := FALSE;
      SPARE_4 : Bool := FALSE;
      SPARE_5 : Bool := FALSE;
      SPARE_6 : Bool := FALSE;
      SPARE_7 : Bool := FALSE;
      SPARE_8 : Bool := FALSE;
      SPARE_9 : Bool := FALSE;
      SPARE_10 : Bool := FALSE;
      "SEPA UW IONIZER TOP MAINTERNANCE DETECTION" : Bool := FALSE;
      "SEPA UW IONIZER TOP DISCHARGE STOP" : Bool := FALSE;
      SPARE : Bool := FALSE;
      SPARE_1 : Bool := FALSE;
      "SEPA UW IONIZER BOTTOM MAINTERNANCE DETECTION" : Bool := FALSE;
      "SEPA UW IONIZER BOTTOM DISCHARGE STOP" : Bool := FALSE;
   END_VAR
BEGIN
END_DATA_BLOCK

